# B&R Automation Studio project x20ost (part 2)

#### bnrcomserver.c
```c
/********************************************************************
 * COPYRIGHT -- Kontora
 ********************************************************************
 * Program: bnrmain
 * File: bnrlsens.c
 * Author: Abramenya
 * Created: January 19, 2009
 *******************************************************************/

#include "bnrcomserver.h"
#ifdef _DEFAULT_INCLUDES
 #include <AsDefault.h>
#endif
//extern SINT *chPortType[];
//extern SINT *chPortRate[];
extern WORD m_wPhoneKey;
extern char StrPhone[50];
/*
DEV_ARM_PORT_TCP=0,
DEV_ARM_PORT_UDP,
DEV_ARM_PORT_COM232,
DEV_ARM_PORT_COM458,
DEV_ARM_PORT_USB,
DEV_SYS_INTERFACE,
*/
SINT *chPortType[] =
{
	"TCP",
	"UDP",
	"RS232",
	"RS485",
	"USB",
};
SINT *chPortRate[] =
{
    "9600",
    "14400",
    "38400",
    "57600",
    "115200",
};
SINT *chPortParity[] =
{
    "N",
	"E",
	"O",
};
SINT *chPortData[] =
{
    "7",
	"8",
};
SINT *chPortStop[] =
{
    "1",
    "1.5",
    "2",
};
SINT *chTest = {"000=1.23000=2.30400=5.60005=192.10000=12334.20001=423.20001=4342.20"};
///char test={'000=0.00000=0.00000=0.00000=0.00000=0.00000=0.}
_GLOBAL UINT node_nr;
_GLOBAL UDINT status;
_GLOBAL CANopen_typ CANopen_01;
_GLOBAL CANnode_typ CANnode_01;
_GLOBAL  FRM_xopen_typ m_sXOpen;
_GLOBAL      XOPENCONFIG m_sConfig;
_GLOBAL      FRM_gbuf_typ m_sFrameBuff;
_GLOBAL      FRM_rbuf_typ m_sRBuff;
_GLOBAL      FRM_write_typ m_sSend;
_GLOBAL 	 FRM_read_typ m_sRecc;
_GLOBAL 	 FRM_close_typ m_sClose;
_GLOBAL 	 FRM_robuf_typ m_sRobuff;
#ifndef WIN32
_GLOBAL      FRM_mode_typ FrameModeStruct;
#endif
//USINT m_SendBuffer[300];
	 //USINT m_ReadBuffer[300];
#ifdef WIN32
#define  START_BYTE   0x7E
#define  STOP_BYTE    0xE7
#define  INVERSE_BYTE 0x55
CComServer *m_nCommServer;
BYTE m_byReadBuffer[300];
BYTE m_bySendBuffer[300];
HANDLE hCom;
OVERLAPPED  osReceive, osSend, osOverlap,osOverlapR;
COMSTAT  csStat;
HANDLE  hSendThread,hSendMsgThread,hReceiveThread,hMakeThread;
HANDLE  WaitEvents[2],evMake;
DWORD   dSendThreadId,dMakeThreadId,dSendMsgThreadId,dReceiveThreadId;
DWORD   dwThrdParam;
void RxCharProc(void);
static DWORD WINAPI SendRsThread(LPVOID lpCComm);
static DWORD WINAPI SendMsgThread(LPVOID lpCComm);
static DWORD WINAPI MakeThread(LPVOID lpCComm);
BOOL OpenPort(char *szComPort, DWORD dwBaud);
BOOL StartPort(char *szPortStr,DWORD dwBaud);
BOOL OpenPort(char *szComPort, DWORD dwBaud)
{
	DCB     dcb;
	COMMTIMEOUTS  ctCom;
	LPSTR lpMsgBuf;
	char  S[100];
	memset(&dcb,0,sizeof(DCB));
	dcb.DCBlength = sizeof(DCB);
    hCom = CreateFile(szComPort,
		GENERIC_READ | GENERIC_WRITE,
		0,
		NULL,
		OPEN_EXISTING,
		FILE_FLAG_OVERLAPPED,
		NULL);
    if (hCom == INVALID_HANDLE_VALUE)
		// ошибка открытия порта
    {
        FormatMessage(
            FORMAT_MESSAGE_ALLOCATE_BUFFER | FORMAT_MESSAGE_FROM_SYSTEM,
            NULL,
            GetLastError(),
            MAKELANGID(LANG_NEUTRAL, SUBLANG_DEFAULT), // Default language
            (LPTSTR) &lpMsgBuf,
            0,
            NULL
			);
        strcpy(S, "Error Opening. ");
        strcat(S, lpMsgBuf);
		printf("\n(__)Com::>%s",S);
		//Info("\n(__)Com::>%s",);
        //MessageBox(NULL, S, "RS232.Open", MB_OK);
        LocalFree( lpMsgBuf );
        return FALSE;
    }
    if (!GetCommState(hCom, &dcb))
		// ошибка получения параметров DCB
    {
        //MessageBox(NULL," Ошибка получения параметров DCB", "RS232.Open", MB_OK);
		printf("\n(__)Com::>Error Get Patrameters DCB");
        CloseHandle(hCom);
        return FALSE;
    }
    dcb.BaudRate = dwBaud;
    dcb.ByteSize = 8;
    dcb.Parity   = NOPARITY;
	//dcb.Parity   = EVENPARITY;
    dcb.StopBits = ONESTOPBIT;
	dcb.fDtrControl = DTR_CONTROL_HANDSHAKE;
	dcb.fRtsControl = RTS_CONTROL_HANDSHAKE;
    //dcb.EvtChar  = (CHAR)STOP_BYTE;
    if (!SetCommState(hCom, &dcb))
		// ошибка установки параметров DCB
    {
        //MessageBox(NULL," Ошибка установки параметров DCB", "RS232.Open", MB_OK);
		printf("\n(__)Com::>Error Create State DCB");
        CloseHandle(hCom);
        return FALSE;
    }
    ctCom.ReadIntervalTimeout = 10;
    ctCom.ReadTotalTimeoutMultiplier  = ctCom.ReadTotalTimeoutConstant  = 1;
    ctCom.WriteTotalTimeoutMultiplier = ctCom.WriteTotalTimeoutConstant = 1;
    if (!SetCommTimeouts(hCom, &ctCom))
		// ошибка установки параметров COMMTIMEOUTS
    {
        //MessageBox(NULL," Ошибка установки параметров COMMTIMEOUTS", "RS232.Open", MB_OK);
		printf("\n(__)Com::>Error DCB");
        CloseHandle(hCom);
        return FALSE;
    }
    //if (!SetCommMask(hCom, EV_RXCHAR|EV_TXEMPTY))
	if (!SetCommMask(hCom, EV_TXEMPTY))
		//    if (!SetCommMask(hCom, EV_BREAK | EV_RXCHAR))
		// ошибка установки маски событий
    {
		printf("\n(__)Com::>Error Create Mask Events");
        CloseHandle(hCom);
        return FALSE;
    }
    PurgeComm(hCom, PURGE_TXCLEAR | PURGE_RXCLEAR);
    // COM-порт успешно открыт и инициализирован
    return TRUE;
}
BOOL StartPort(char *szPortStr,DWORD dwBaud)
{
	if (OpenPort(szPortStr, dwBaud) != TRUE)
	{
		return FALSE;
	}
	if ((osOverlap.hEvent = CreateEvent(NULL, FALSE, FALSE, NULL)) == NULL)
	{
		printf("\n(__)Com::> Error Create osOverlap.hEvent");
		return FALSE;
	}

	if ((osReceive.hEvent = CreateEvent(NULL, FALSE, FALSE, NULL)) == NULL)
	{
		printf("\n(__)Com::> Error Create osReceive.hEvent");
		return FALSE;
	}
	if ((osSend.hEvent = CreateEvent(NULL, FALSE, FALSE, NULL)) == NULL)
	{
		printf("\n(__)Com::> Error Create osSend.hEvent");
		return FALSE;
	}
	if ((evMake = CreateEvent(NULL, FALSE, FALSE, NULL)) == NULL)
	{
		printf("\n(__)Com::> Error Create evMake");
		return FALSE;
	}
	if ((hMakeThread = CreateThread(NULL,0,MakeThread,&dwThrdParam,0,&dMakeThreadId)) == NULL)
	{
		printf("\n(__)Com::> Error Create hMakeThread");
		return FALSE;
	}
	if ((hSendThread = CreateThread(NULL,0,SendRsThread,&dwThrdParam,0,&dSendThreadId)) == NULL)
	{
		printf("\n(__)Com::> Error Create hReceiveThread");
		return FALSE;
	}

	if ((hSendMsgThread = CreateThread(NULL,0,SendMsgThread,&dwThrdParam,0,&dSendMsgThreadId)) == NULL)
	{
		printf("\n(__)Com::> Error Create hSensMsgThread");
		return FALSE;
	}
	SetThreadPriority(hSendThread, THREAD_PRIORITY_HIGHEST);
	SetThreadPriority(hSendMsgThread, THREAD_PRIORITY_NORMAL);
	SetThreadPriority(hMakeThread, THREAD_PRIORITY_NORMAL);
	ResumeThread(hSendThread);
	ResumeThread(hSendMsgThread);
	ResumeThread(hMakeThread);
	return TRUE;
}
void ClosePort(void)
{
    if (hCom != INVALID_HANDLE_VALUE)
    {
      CloseHandle(hCom);
      hCom = INVALID_HANDLE_VALUE;
    }
}
DWORD WINAPI SendMsgThread(LPVOID lpCComm)
{
    while(1)
    {
      m_nCommServer->SendThread(m_nCommServer);
	  Sleep(100);
    }
}
DWORD WINAPI SendRsThread(LPVOID lpCComm)
{
	DWORD dwMask,dwBytesTrans;
	//SMESSAGE mMsg;
	while(1)
	{
      //printf("\n(__)Com::>SendRsThread");
	  WaitCommEvent(hCom,&dwMask,&osOverlap);
	  //switch (WaitForSingleObject(osOverlap.hEvent,INFINITE))
	  switch (WaitForSingleObject(osOverlap.hEvent,5000))
	  {
	    case WAIT_OBJECT_0:
			 if (GetOverlappedResult(hCom,&osOverlap,&dwBytesTrans,TRUE))
			 {
               if (dwMask&EV_TXEMPTY)
               {
                //printf("\n(__)Com::>EV_TXEMPTY");
				m_sSend.status = 0;
				m_nCommServer->m_StatusWrite = 0;
               }
			   if (dwMask&EV_RXCHAR)
               {
				//printf("\n(__)Com::>EV_RXCHAR");
				//m_nCommServer->ReceiveThread(m_nCommServer);
				//RxCharProc();
               }
			 }
	  	break;
		case WAIT_TIMEOUT:
			 m_sSend.status = 0;
			 m_nCommServer->m_StatusWrite = 0;
			 PurgeComm(hCom, PURGE_TXCLEAR | PURGE_RXCLEAR);
			 //printf("\n(__)Com::>TX:WAIT_TIMEOUT");
		break;
	  }
	  //Sleep(1);
	}
}
void FRM_xopen(FRM_xopen_typ *pType)
{
    StartPort("COM4",1200);
};
void FRM_close(FRM_close_typ *pType){};
void FRM_gbuf(FRM_gbuf_typ *pType)
{
	pType->status = 0;
	pType->buflng = 300;
	pType->buffer = &m_bySendBuffer[0];
};
void FRM_rbuf(FRM_rbuf_typ *pType){};
void FRM_robuf(FRM_robuf_typ *pType){};
char chBuff[100];
void FRM_write(FRM_write_typ *pType)
{
	DWORD dwSentBytes;
	BOOL res;
	pType->status = 1;
	m_nCommServer->m_StatusWrite = 1;
	if(!WriteFile(hCom, pType->buffer, pType->buflng, &dwSentBytes,&osSend))
	//strcpy(chBuff,"Abramenya Alex");
	//if(!WriteFile(hCom, chBuff, strlen(chBuff), &dwSentBytes,&osOverlap))
    {
     if(GetLastError() != ERROR_IO_PENDING)
     {
	  // Ошибка записи данных
      res = FALSE;
	  printf("\n(__)Com::>Write Error 0.");
     }else
     {
      if(!GetOverlappedResult(hCom, &osSend, &dwSentBytes, TRUE))
      {
	   printf("\n(__)Com::>Write Error 1.");
      }else
      {
	   // Запись данных закончена
       res = TRUE;
	   //pType->status = 1;
	   //m_nCommServer->m_StatusWrite = 1;
	   //printf("\n(__)Com::>Write Ok 0.");
      }
     }
    }
    else
    {
	 // Запись успешно завершена
     res = TRUE;
	 //printf("\n(__)Com::>Write Ok 1.");
    }
};
BYTE pb_mBoxDoRead[5000];
BYTE pb_mBoxRead[3000];
BYTE pb_mBoxCont[5000];
WORD w_mBoxSize  = 0x7ff;
WORD w_mBoxCSize = 0x7ff;
WORD w_mBoxWrite = 0;
WORD w_mBoxRead  = 0;
WORD w_mBoxMesCt = 0;
//WORD w_mBoxSEnd  = 50000;
WORD mCurLen=0;
WORD m_sSize=0;
WORD w_lLength=0;
void MakeMessage(void);
void CopyMessage(WORD wLen);
/*
Success := ReadFile(FHandle, pb_mBoxDoRead, w_lLength, BytesTrans, @Ov);
		 for i:=0 to w_lLength-1 do
		 Begin
		  pb_mBoxCont[w_mBoxWrite]:=pb_mBoxDoRead[i];
          w_mBoxWrite := (w_mBoxWrite + 1) and BSZ;
		  //SendDebug('(__)Synchro Buffer NULL.');
		 End;

			 //SendDebug('(__)RD::');
			 //for i:=0 to w_lLength-1 do SendDebug(' '+IntToStr(pb_mBoxCont[i]));
			 //Success := Success and GetOverlappedResult(FHandle, Ov, BytesTrans, False);
			 //w_mBoxWrite := (w_mBoxWrite + w_lLength)and $7ff;
w_mBoxSize  := w_mBoxSize   - w_lLength;
m_sSize     := w_mBoxCSize  - w_mBoxSize;
			 if ((pb_mBoxCont[w_mBoxRead]=$68)or(pb_mBoxCont[w_mBoxRead]=$10)) then
				 Begin
m_byMType := 0;
			 SetEvent(hRxEvent);
			 End else
				 Begin
m_byMType  := 1;
w_mBoxSize  := BSZ;
w_mBoxCSize := BSZ;
w_mBoxWrite := 0;
w_mBoxRead  := 0;
w_mBoxMesCt := 0;
m_sSize:=0;
FBlTxEmpty := True;
			SendDebug('(__)Synchro Buffer.');
			//SetEvent(hRxEvent);
  End;
*/
void FRM_read(FRM_read_typ *pType)
{
	DWORD Errors,BytesTrans;
	BYTE i;
	ClearCommError(hCom, &Errors, &csStat);
	pType->status = 1;
	if (csStat.cbInQue!=0)
	{
	 pType->buffer = &m_byReadBuffer[0];
	 w_lLength = csStat.cbInQue;
     if(ReadFile(hCom, pType->buffer, w_lLength, &BytesTrans, &osReceive))
	 //if(ReadFile(hCom, m_byReadBuffer, w_lLength, &BytesTrans, &osReceive))
	 {
	  //for(i=0;i<w_lLength-1;i++)printf(" %x",m_byReadBuffer[i]);
	  pType->buflng = w_lLength;
	  pType->status = 0;
	 }else Info("\nError Read_0.");
	}
}
void RxCharProc(void)
{
	DWORD Errors,BytesTrans,dwB;
    BOOL  res;
	INT   i,wI,lLen;
	ClearCommError(hCom, &Errors, &csStat);
	if (csStat.cbInQue!=0)
	{
     w_lLength = csStat.cbInQue;
     if ((w_lLength<=0)||(w_lLength>500)) return;
     wI = w_mBoxWrite;
     if((wI+w_lLength)<=w_mBoxCSize)res = ReadFile(hCom, &pb_mBoxCont[wI], w_lLength, &BytesTrans, &osReceive);else
	 {
      res = ReadFile(hCom, &pb_mBoxDoRead[0], w_lLength, &BytesTrans, &osReceive);
	  for (i=0;i<w_lLength;i++){pb_mBoxCont[wI]=pb_mBoxDoRead[i];wI = (wI + 1) & 0x7ff;}
	 }
	 if(GetOverlappedResult(hCom, &osReceive, &dwB, TRUE))
	 {
	  //printf("\n(__)COM::>");for(i=0;i<w_lLength;i++)printf(" %x",pb_mBoxCont[w_mBoxWrite+i]);

	  w_mBoxWrite = (w_mBoxWrite + w_lLength)& 0x7ff;
      mCurLen=mCurLen+w_lLength;
      w_mBoxSize  = w_mBoxSize  - w_lLength;
	  if ((pb_mBoxCont[w_mBoxRead]==0x68)||(pb_mBoxCont[w_mBoxRead]==0x10))
	  {
       m_sSize=w_mBoxCSize-w_mBoxSize;
       SetEvent(evMake);
	   mCurLen=0;
	  }

	 }else printf("\n(__)Com::>RxRead Error.");
	}
}
void MakeMessage(void)
{
   WORD lLen,i;
   //printf("\n(__)COM::>MAKE_M:%x",pb_mBoxCont[w_mBoxRead]);
   lLen = pb_mBoxCont[(w_mBoxRead+1) & 0x7ff];
   while((m_sSize>=(lLen+6))&&(pb_mBoxCont[w_mBoxRead]==0x68))CopyMessage(lLen+6);
   lLen = 5;
   while((m_sSize>=lLen)&&(pb_mBoxCont[w_mBoxRead]==0x10))CopyMessage(lLen);
}
void CopyMessage(WORD wLen)
{
   INT i;
   SMESSAGE sMsg;
   for(i=0;i<wLen;i++)
   {
    pb_mBoxRead[i]=pb_mBoxCont[w_mBoxRead];
    w_mBoxSize++;
    w_mBoxRead=(w_mBoxRead+1)& 0x7ff;
   }
   m_sSize = (w_mBoxCSize-w_mBoxSize) & 0x7ff;
   m_sRecc.buflng = wLen;
   memcpy(&m_byReadBuffer[0],pb_mBoxRead, wLen);
   m_nCommServer->ReceiveThread(m_nCommServer);
   //printf("\n(__)COM::>");for(i=0;i<wLen;i++) printf(" %x",pb_mBoxRead[i]);
}
DWORD WINAPI MakeThread(LPVOID lpCComm)
{
	BYTE i;
	 while(1)
	 {
      WaitForSingleObject(evMake,INFINITE);
	  MakeMessage();
	  //printf("\n(__)COM::>MakeM.");
	 }
}
void CANopen(CANopen_typ *pCANOpen){};
void CANnode(CANnode_typ *pCANnode){};
#endif

void CComServer_Init(This,SARMINTERFACE *pArm)
{
    DECLARE_MULTI_OPEN(CComServer,CCyclicSystem)
    #ifdef WIN32
	m_nCommServer = pT;
    #endif
	pT->m_pArm = pArm;
	FDEFINE(DEV_RSMMD_BOX_ID,DEV_RSMMD_BOX_SZ);
	FDEFINE(DEV_RSBUF_BOX_ID,DEV_RSBUF_BOX_SZ);
	pB->SetBoxID(pB,DEV_RSMMD_BOX_ID);

	InitObject(CMTimer,&pT->m_nConnTMR);
	pT->m_nConnTMR.SetTimer(&pT->m_nConnTMR,DIR_PHTOPH,DIR_PHTOPH,EV_TMR_SRR_REQ,0,0,DEV_RSMMD_BOX_ID);
	//pT->m_nConnTMR.OnTimer(&pT->m_nConnTMR,10);
	pT->m_blMsgFind = FALSE;
	pT->m_byType = pArm->byType;
	pT->m_byRate = pArm->byPortRate;
	pT->InByteCount_DATA = 0;

	strcpy(pT->m_chStringMode, chPortType[pT->m_pArm->byType]);
	strcat(pT->m_chStringMode,", ");
	strcat(pT->m_chStringMode, chPortRate[pT->m_pArm->byPortRate]);
	strcat(pT->m_chStringMode,", ");
	strcat(pT->m_chStringMode, chPortParity[pT->m_pArm->stTcpAddr.byAddr0]);
	strcat(pT->m_chStringMode,", ");
	strcat(pT->m_chStringMode, chPortData[pT->m_pArm->stTcpAddr.byAddr1]);
	strcat(pT->m_chStringMode,", ");
	strcat(pT->m_chStringMode, chPortStop[pT->m_pArm->stTcpAddr.byAddr2]);

	strcpy(pT->m_chStringDevice, "SL0.IF1");
	#ifdef DEB_CComServer
	Info("\n(__)CTCPS::>Create %s.Device: %s Mode: %s",
	chPortType[pT->m_byType],pT->m_chStringDevice,pT->m_chStringMode);
	#endif
	pT->SynBuff(pT);
    pT->InitSRV(pT);
	//pT->m_nConnTMR.OnTimer(&pT->m_nConnTMR,200);
	pT->m_StatusWrite = 0;
	pT->m_bSrvState = DRV_ST_CONN;
	pT->m_bCliState = DRV_ST_CONN;
}
/*
if(pA->byA2==0) pR->byNumber          = (BYTE)pA->wParam; //Port Number
if(pA->byA2==1) pR->byType            = (BYTE)pA->wParam; //Port Type
if(pA->byA2==2) pR->byPortRate        = (BYTE)pA->wParam; //Port Rate
if(pA->byA2==3) pR->stTcpAddr.byAddr0 = (BYTE)pA->wParam; //Parity
if(pA->byA2==4) pR->stTcpAddr.byAddr1 = (BYTE)pA->wParam; //Data Bits
	 if(pA->byA2==5) pR->stTcpAddr.byAddr2 = (BYTE)pA->wParam; //Stop Bits
*/
void CComServer_SetPortSett(This)
{
    DECLARE_MULTI_OPEN(CComServer,CCyclicSystem)
    strcpy(pT->m_chStringDevice, "SL0.IF1");
	memset(pT->m_chStringNewMode,0,sizeof(pT->m_chStringNewMode));

	strcpy(pT->m_chStringNewMode, chPortType[pT->m_pArm->byType]);
	strcat(pT->m_chStringNewMode,", ");
	strcat(pT->m_chStringNewMode, chPortRate[pT->m_pArm->byPortRate]);
	strcat(pT->m_chStringNewMode,", ");
	strcat(pT->m_chStringNewMode, chPortParity[pT->m_pArm->stTcpAddr.byAddr0]);
	strcat(pT->m_chStringNewMode,", ");
	strcat(pT->m_chStringNewMode, chPortData[pT->m_pArm->stTcpAddr.byAddr1]);
	strcat(pT->m_chStringNewMode,", ");
	strcat(pT->m_chStringNewMode, chPortStop[pT->m_pArm->stTcpAddr.byAddr2]);
    #ifndef WIN32
    FrameModeStruct.ident  = m_sXOpen.ident;
    FrameModeStruct.mode   = (UDINT)pT->m_chStringNewMode;
    FrameModeStruct.enable = 1;
    FRM_mode(&FrameModeStruct);
    #endif
}
void CComServer_SynBuff(This)//CANOpen
{
    DECLARE_MULTI_OPEN(CComServer,CCyclicSystem)
	pT->w_mBoxSize  = BUFF_SZ;
    pT->w_mBoxCSize = BUFF_SZ;
	pT->w_mBoxWrite = 0;
	pT->w_mBoxRead  = 0;
	pT->m_sSize     = 0;
	pT->w_lLength   = 0;
	pT->w_lMsgLen   = 0;
	memset(&pT->pb_mBoxCont[0],0,10);
	#ifdef DEB_CComServer
	Info("\n(__)CTCPS::>Synchro.");
    #endif
}
_GLOBAL FRM_xopen_typ FrameXOpenStruct;
_GLOBAL XOPENCONFIG XOpenConfigStruct;
void CComServer_InitSRV(This)
{
    DECLARE_MULTI_OPEN(CComServer,CCyclicSystem)

	CANopen_01.enable    = 1;
    CANopen_01.baud_rate = 25;
    CANopen_01.cob_anz   = 5;
    CANopen_01.device    = 0;
    CANopen(&CANopen_01);

	//Server Init
    m_sConfig.idle     = 10;
    m_sConfig.delimc   = 0;
    m_sConfig.delim[0] = 0;
	m_sConfig.delim[1] = 0;
	m_sConfig.tx_cnt   = 2;
	m_sConfig.rx_cnt   = 2;
	m_sConfig.tx_len   = 256;
	m_sConfig.rx_len   = 256;
	m_sConfig.argc     = 0;
	m_sConfig.argv     = 0;

	strcpy(pT->m_chStringMode, "RS232, 57600, E, 8, 1");
	m_sXOpen.device    = (UDINT) pT->m_chStringDevice;
	m_sXOpen.mode      = (UDINT) pT->m_chStringMode;
    m_sXOpen.config    = (UDINT)&m_sConfig;
	m_sXOpen.enable    = 1;
	pT->m_StatusOpen   = 0;
    #ifndef WIN32
	pT->m_nConnTMR.OnTimer(&pT->m_nConnTMR,30);
    #else
	pT->m_nConnTMR.OnTimer(&pT->m_nConnTMR,30);
	//pT->Open(pT);
    #endif
}
_GLOBAL INT nOPEN,nCLOSE;

BOOL CComServer_Open(This)
{
    DECLARE_MULTI_OPEN(CComServer,CCyclicSystem)
	SHORTMESSAGE m_sMsg;

	CANnode_01.enable = 1;
    CANnode(&CANnode_01);
    node_nr = CANnode_01.node_nr;
    #ifdef WIN32
	node_nr = 1;
	//pT->m_StatusOpen = 0;
    #endif
    if((node_nr==1)&&(pT->m_StatusOpen==0))
	{
	FRM_xopen(&m_sXOpen);
	if(m_sXOpen.status==0)
	{
	 nOPEN++;
	 m_sRecc.ident      = m_sXOpen.ident;
	 m_sSend.ident      = m_sXOpen.ident;
	 m_sClose.ident     = m_sXOpen.ident;
	 m_sFrameBuff.ident = m_sXOpen.ident;
	 m_sRBuff.ident     = m_sXOpen.ident;
	 m_sRecc.buffer	    = (UDINT)&pT->m_ReadBuffer[0];
	 m_sSend.buffer     = (UDINT)&pT->m_SendBuffer[0];
	 m_sFrameBuff.buffer= m_sSend.buffer;
	 m_sRBuff.buffer    = m_sRecc.buffer;
	 m_sRecc.enable     = 1;
	 m_sSend.enable     = 1;
	 m_sClose.enable    = 1;
	 m_sFrameBuff.enable= 1;
	 m_sRBuff.enable    = 1;
	 pT->m_StatusOpen   = 1;
	 pT->m_StatusWrite  = 0;
     #ifdef IF_MODEM
	 SendCommand(PH_INIT_REQ,"AT+ipr=57600");
	 SendCommand(PH_INIT_REQ,"AT+icf=2,1");
	 SendCommand(PH_INIT_REQ,"AT+ifc=0,0");
	 SendCommand(PH_INIT_REQ,"AT&D1");
	 SendCommand(PH_INIT_REQ,"AT&C1");
	 //SendCommand(PH_INIT_REQ,"AT&S0");
	 SendCommand(PH_INIT_REQ,"ATS0=1");
	 SendCommand(PH_INIT_REQ,"AT+CLIP=1");
     #endif
	 pT->SendSMessage(pT,DEV_KPMDL_BOX_ID,DIR_PHTOKP,PH_CALL_REQ);
	 return TRUE;
	}
 	}
	if((node_nr==3)&&(pT->m_StatusOpen==1))
	{
	  nCLOSE++;
	  pT->m_StatusOpen = 0;
      pT->Close(pT);
	  return TRUE;
	}
	return FALSE;
}
void CComServer_Enable(This)
{
	DECLARE_MULTI_OPEN(CComServer,CCyclicSystem)
	m_sXOpen.enable = 1;
}
void CComServer_Disable(This)
{
	DECLARE_MULTI_OPEN(CComServer,CCyclicSystem)
	m_sXOpen.enable = 0;
}
void CComServer_Close(This)
{
    DECLARE_MULTI_OPEN(CComServer,CCyclicSystem)
	m_sClose.enable = 1;
	FRM_close(&m_sClose);
}
BOOL CComServer_SendMessage(This,SMESSAGE *pMsg)
{
	DECLARE_MULTI_OPEN(CComServer,CCyclicSystem)
	BOOL res = TRUE;
	if(pT->m_StatusOpen==1)
	{
	 FRM_gbuf(&m_sFrameBuff);
     m_sSend.buflng = pMsg->m_swLen-9;
	 memcpy(m_sSend.buffer, &pMsg->m_sbyInfo[0],m_sSend.buflng);
	 FRM_write(&m_sSend);
	 pT->m_StatusWrite  = m_sSend.status;
	 if(pT->m_StatusWrite==0) res = TRUE;else res = FALSE;
	}
	return res;
}
_GLOBAL INT nSND;
_GLOBAL INT nSendThread;
void CComServer_SendThread(This)
{
    DECLARE_MULTI_OPEN(CComServer,CCyclicSystem)
	nSendThread++;
    //if(pT->m_StatusWrite==0)
	if(pT->m_StatusOpen==1)
    {
	 #ifdef DEB_CComServer
	 //pT->TestMsg(pT);
     #endif
	 if(FGET(DEV_RSBUF_BOX_ID,&pT->m_sMsg))
	 {
	  //Info("\n(__)CRSSM::>TX:%M",&pT->m_sMsg);
	  if(pT->m_sMsg.m_swLen<=256)
	  {
	   nSND++;
       pT->SendMessage(pT,&pT->m_sMsg);
	  }//else
	    //Info("\n(__)CRSSM::>Wery Long Message!");
	 }
	}
}
_GLOBAL INT nGETL1;
BOOL CComServer_GetMessage(This,SMESSAGE *pMsg)
{
    DECLARE_MULTI_OPEN(CComServer,CCyclicSystem)
	BYTE i,*pBuff;
	BOOL res=FALSE;
	SMESSAGE csM;
	if(pT->m_StatusOpen==1)
	{
	FRM_read(&m_sRecc);
	pT->m_StatusRead       = m_sRecc.status;
	if(pT->m_StatusRead==0)
	{
	 pT->m_ReadBufferLength = m_sRecc.buflng;
	 pBuff                  = m_sRecc.buffer;
	 /*
	 csM.m_sbyInfo[0] = 0x7e;
	 csM.m_sbyInfo[1] = 'A';
	 csM.m_sbyInfo[2] = 'l';
	 csM.m_sbyInfo[3] = 'e';
	 csM.m_sbyInfo[4] = 'x';
	 csM.m_sbyInfo[5] = 'a';
	 csM.m_sbyInfo[6] = 'n';
	 csM.m_sbyInfo[7] = 'd';
	 csM.m_sbyInfo[8] = 'e';
	 csM.m_sbyInfo[9] = 'r';
	 csM.m_sbyInfo[10] = 0xe7;
	 */

	 //memcpy(&csM.m_sbyInfo[0],m_sRecc.buffer,pT->m_ReadBufferLength);
	 //csM.m_swLen = 9 + pT->m_ReadBufferLength;
	 //Info("\n(__)CRSSM::>MSG:%M",&csM);

	 //m_sRBuff.buffer = m_sRecc.buffer;
	 //m_sRBuff.buflng = pT->m_ReadBufferLength;
	 //FRM_rbuf(&m_sRBuff);
	 //res = TRUE;
	 //nGETL1++;
	 //Info("\nMSG::>");
	 //csM.m_swLen = pT->m_ReadBufferLength+9;
	 for( i=0;i<pT->m_ReadBufferLength;i++)
	 {
	  pT->pb_mBoxCont[pT->w_mBoxWrite] = pBuff[i];
      //Info(" %b",&pT->pb_mBoxCont[pT->w_mBoxWrite]);
	  //printf(" %c",pT->pb_mBoxCont[pT->w_mBoxWrite]);
      pT->w_mBoxWrite = (pT->w_mBoxWrite + 1) & BUFF_SZ;
	 }
	 //FPUT(DEV_RSBUF_BOX_ID,(BYTE*)&csM);
	 pT->w_mBoxSize -= pT->m_ReadBufferLength;
	 pT->m_sSize     = pT->w_mBoxCSize-pT->w_mBoxSize;
	 //Info("\nRD::>%b PRD::>%w PWD::>%w FND::>%b",&pT->pb_mBoxCont[pT->w_mBoxRead],&pT->w_mBoxRead,&pT->w_mBoxWrite,&pT->m_blMsgFind);
	 //printf(" %c %c", pT->pb_mBoxCont[pT->w_mBoxRead],pT->pb_mBoxCont[pT->w_mBoxRead+1]);
	 //if ((pT->pb_mBoxCont[pT->w_mBoxRead]==0x3d)&&(pT->pb_mBoxCont[pT->w_mBoxRead+1]==0x30))
	 if ((pT->pb_mBoxCont[pT->w_mBoxRead]==0x3d))
	 {
	  pT->m_blMsgFind = TRUE;
	  if(res = pT->MakeMsgData(pT,pMsg))
	  {
	   pT->m_blMsgFind = FALSE;
	   res = TRUE;
	  }
	 }else
		 pT->SynBuff(pT);
	 //if (pT->m_blMsgFind==FALSE)
	 //{
	 //	pT->MakeTextMessage(pT);
 	 //}else /*if (pT->pb_mBoxCont[pT->w_mBoxRead]==0x41)*/ pT->SynBuff(pT);
	 m_sRBuff.buffer = m_sRecc.buffer;
	 m_sRBuff.buflng = pT->m_ReadBufferLength;
	 FRM_rbuf(&m_sRBuff);
     }
	}
	return res;
}
BOOL CComServer_MakeMsgData(This,SMESSAGE *pMsg)
{
    DECLARE_MULTI_OPEN(CComServer,CCyclicSystem)
	WORD lLen,i,nCM=0;
	BOOL res = FALSE;
	lLen = 1;
	pT->w_lMsgLen = pT->w_lMsgLen + pT->m_ReadBufferLength;
	if (pT->w_lMsgLen>BUFF_SZ) {pT->SynBuff(pT);return res;}
    for (i=1;i<pT->w_lMsgLen-1;i++)
	{
	 lLen++;
	 if (pT->pb_mBoxCont[(pT->w_mBoxRead+i)& BUFF_SZ]==0x2e) nCM++;
	 if (nCM>1){pT->SynBuff(pT);return res;}
	 if (lLen>300) {pT->SynBuff(pT);return res;}
     if (pT->pb_mBoxCont[(pT->w_mBoxRead+i)& BUFF_SZ]==0x3d)
     {
	  pT->CopyMessage(pT,lLen,pMsg);
	  //pT->SynBuff(pT);
	  pT->w_lMsgLen = 0;
	  return TRUE;
	 }
	}
	return res;
}
BOOL CComServer_CopyMessage(This,WORD wLen,SMESSAGE *pMsg)
{
    DECLARE_MULTI_OPEN(CComServer,CCyclicSystem)
    INT i,j=0;BYTE byCRC;
	BOOL blCRC;
	for(i=0;i<wLen;i++)
	{
	 if ((i!=0)&&(i!=wLen-1)){pMsg->m_sbyInfo[j]=pT->pb_mBoxCont[pT->w_mBoxRead];j++;}
	 pT->w_mBoxSize =(pT->w_mBoxSize+1)& BUFF_SZ; ;
	 pT->w_mBoxRead=(pT->w_mBoxRead+1)& BUFF_SZ;
	 //Info(" %b",&pMsg->m_sbyInfo[i]);
	 //printf(" %x",pMsg->m_sbyInfo[i]);
	}
	pMsg->m_sbyInfo[j++] = 0x00;
	pT->w_mBoxRead=(pT->w_mBoxRead-1)& BUFF_SZ;
	pT->m_sSize = (pT->w_mBoxCSize-pT->w_mBoxSize) & BUFF_SZ;
	pMsg->m_swLen         = j+9;
	pMsg->m_sbyFrom       = DIR_PHMDL;
	pMsg->m_sbyFor        = DIR_PHTOMS;
	pMsg->m_sbyIntType    = 0;
	pMsg->m_sbyServerID   = 0;
	pMsg->m_sbyType       = PH_VS0_REQ;
	pMsg->m_sbyDirection  = 0;
	pMsg->m_sbySensor     = 0;
	//byCRC = pMsg->m_sbyInfo[pMsg->m_swLen-9-2];
    //if (pMsg->m_sbyInfo[0]==MSG_SHRT_CODE)
	//if (byCRC==pT->CreateCRC(pT,&pMsg->m_sbyInfo[1],2)) blCRC = TRUE;
	return TRUE;
}
_GLOBAL INT nReceiveThread;
void CComServer_ReceiveThread(This)
{
    DECLARE_MULTI_OPEN(CComServer,CCyclicSystem)
	nReceiveThread++;
	if(pT->GetMessage(pT,&pT->m_sMsg)==TRUE)
	{
	 //Info("\n(__)CRSSM::>RX:%M",&pT->m_sMsg);
	 //if ((pT->nWsCount++)%10==0)
	 FPUT(DEV_MSMDL_BOX_ID,(BYTE*)&pT->m_sMsg);
	 //FPUT(DEV_RSBUF_BOX_ID,(BYTE*)&pT->m_sMsg);
	}
}
void CComServer_MakeTextMessage(This)
{
	DECLARE_MULTI_OPEN(CComServer,CCyclicSystem)
    BYTE byInByte;
    while (pT->w_mBoxWrite!=pT->w_mBoxRead)
	{
     byInByte = pT->pb_mBoxCont[pT->w_mBoxRead];
     pT->w_mBoxRead = (pT->w_mBoxRead+1) & BUFF_SZ;
     if (pT->w_mBoxSize>pT->w_mBoxCSize){pT->SynBuff(pT);return;};
     pT->w_mBoxSize++;
     if (byInByte==0x0d)
	 {
	   if (pT->InByteCount_DATA>1)
	   pT->ATHandler(pT,&pT->pb_mBoxDoTextRead[0],pT->InByteCount_DATA);
       pT->InByteCount_DATA = 0;
	 }else
	 {
       pT->pb_mBoxDoTextRead[pT->InByteCount_DATA] = byInByte;
       if (pT->InByteCount_DATA>100) {pT->InByteCount_DATA=0;pT->SynBuff(pT);}
       pT->InByteCount_DATA++;
	 }
	}
}
void CComServer_ATHandler(This,USINT *pComm,WORD wLen)
{
    DECLARE_MULTI_OPEN(CComServer,CCyclicSystem)
    WORD i,i0,i1,j=0;
	//printf("\nAT_MSG::>");for (i=0;i<wLen;i++)printf(" %c",pComm[i]);
	if (wLen<100)
	{
	pComm[wLen] = 0;
	if(pT->FindText(pT,"CONNECT",pComm)>0)
	{
     #ifdef DEB_CComServer
	 Info("\n(__)CRSSM::>CONNECT 9600");
     #endif
	 pT->Connect(pT);
	 return;
	}
	if(pT->FindText(pT,"NO CAR",pComm)>0)
	{
     #ifdef DEB_CComServer
	 Info("\n(__)CRSSM::>NO CARRIER");
     #endif
	 pT->Disconnect(pT);
	 return;
	}
	if(pT->FindText(pT,"+CLIP:",pComm)>0)
	{
     #ifdef DEB_CComServer
	 Info("\n(__)CRSSM::>+CLIP");
     #endif
     m_wPhoneKey = 0;
	 i0 = pT->FindText(pT," ",pComm);i1 = pT->FindText(pT,",",pComm);
     //printf("\nAT_PHO::>");
	 for (i=i0+2;i<i1-1;i++)
	 {
	  if (i>30) return;
	  m_wPhoneKey = m_wPhoneKey + ((pComm[i]&0x0f)+j);
	  //StrPhone[j]=pComm[i];
	  j++;
      //printf(" %c",pComm[i]);
	 }
	 return;
	}
	}else pT->SynBuff(pT);
}
INT CComServer_FindText(This,SINT *pSrc,SINT *pChar)
{
    DECLARE_MULTI_OPEN(CComServer,CCyclicSystem)
	WORD i,wSrcSumm=0,wLen,wStrLen;
	wLen    = strlen(pSrc);
	wStrLen = strlen(pChar);
	wSrcSumm = pT->CalckSumm(pT,(BYTE*)pSrc,wLen);
	for (i=0;i<wStrLen-wLen;i++)
	{
	 if (wSrcSumm==pT->CalckSumm(pT,(BYTE*)&pChar[i],wLen))
	 return i;
	}
	return -1;
}
WORD CComServer_CalckSumm(This,BYTE *pCH,WORD wLen)
{
    DECLARE_MULTI_OPEN(CComServer,CCyclicSystem)
	WORD i,wSrcSumm=0;
	for (i=0;i<wLen;i++)
	wSrcSumm += pCH[i];
    return wSrcSumm;
}
BYTE CComServer_CreateCRC(This,BYTE *pMsg,BYTE byLen)
{
	DECLARE_MULTI_OPEN(CComServer,CCyclicSystem)
	BYTE i,sum = 0;
	for(i=0;i<=byLen-1;i++)sum += pMsg[i];
	return sum;
}
_GLOBAL INT nRSEventHandler,nCheckOpen,nWatchOpen;
BOOL CComServer_EventHandler(This,SMESSAGE *pMsg)
{
    DECLARE_MULTI_OPEN(CComServer,CCyclicSystem)
	switch(pMsg->m_sbyFor)
	{
	  case DIR_101TOPH:
	       #ifdef DEB_CComServer
		   //Info("\n(__)CRSSM::>OUTP::%M",pMsg);
		   #endif
		   FPUT(DEV_RSBUF_BOX_ID,pMsg);
	  break;
	  case DIR_KPTO101:
	       nRSEventHandler++;
		   if(pMsg->m_sbyType==PH_CONN_REQ)
		   {
            #ifndef IF_MODEM
		    pT->Connect(pT);
            #else
		    FPUT(DEV_RSBUF_BOX_ID,pMsg);
            #endif
		   }
		   if((pMsg->m_sbyType==PH_DISC_REQ)||(pMsg->m_sbyType==PH_DISC0_REQ))
		   {
			//pT->Disconnect(pT);
			FPUT(DEV_RSBUF_BOX_ID,pMsg);
		   }
		   if(pMsg->m_sbyType==PH_INIT_REQ)
		   FPUT(DEV_RSBUF_BOX_ID,pMsg);
	  break;
	  case DIR_PHTOPH:
	       if (pMsg->m_sbyType==EV_TMR_SRR_REQ)
		   {
		   	//if(pT->m_StatusOpen==0)
			{
			 nCheckOpen++;
 		     pT->Open(pT);
			}
			pT->m_nConnTMR.OnTimer(&pT->m_nConnTMR,30);
		   }
	  break;
      case DIR_KPTOPH:
	       if (pMsg->m_sbyType==PH_CLOSE_PORT_REQ)
		   {
            //pT->Close(pT);
		   }
		   if(pMsg->m_sbyType==PH_INIT_PORT_REQ)
		   {
             pT->SetPortSett(pT);
		   }
	  break;
	  default:
	  break;
	}
	return TRUE;
}
void CComServer_Connect(This)
{
    DECLARE_MULTI_OPEN(CComServer,CCyclicSystem)
    SHORTMESSAGE m_sMsg;
	m_sMsg.m_swLen        = 9;
	m_sMsg.m_sbyFrom      = DIR_PHMDL;
	m_sMsg.m_sbyFor       = DIR_PHTO101P;
	m_sMsg.m_sbyIntType   = 0;
	m_sMsg.m_sbyServerID  = 0;
	m_sMsg.m_sbyType      = PH_CONN_IND;
	m_sMsg.m_sbyDirection = 0;
	m_sMsg.m_sbySensor    = 0;
	FPUT(DEV_101MD_BOX_ID,(BYTE*)&m_sMsg);
    #ifdef DEB_CComServer
	Info("\n(__)CRSSM::>OUTT::%M",&m_sMsg);
    #endif
}
void CComServer_SendSMessage(This,BYTE byBox,BYTE byFor,BYTE byType)
{
    DECLARE_MULTI_OPEN(CComServer,CCyclicSystem)
    SHORTMESSAGE m_sMsg;
	m_sMsg.m_swLen        = 9;
	m_sMsg.m_sbyFrom      = DIR_PHMDL;
	m_sMsg.m_sbyFor       = byFor;
	m_sMsg.m_sbyIntType   = 0;
	m_sMsg.m_sbyServerID  = 0;
	m_sMsg.m_sbyType      = byType;
	m_sMsg.m_sbyDirection = 0;
	m_sMsg.m_sbySensor    = 0;
	FPUT(byBox,(BYTE*)&m_sMsg);
    #ifdef DEB_CComServer
	Info("\n(__)CRSSM::>OUTT::%M",&m_sMsg);
    #endif
}
void CComServer_Disconnect(This)
{
    DECLARE_MULTI_OPEN(CComServer,CCyclicSystem)
    SHORTMESSAGE m_sMsg;
	m_sMsg.m_swLen        = 9;
	m_sMsg.m_sbyFrom      = DIR_PHMDL;
	m_sMsg.m_sbyFor       = DIR_PHTO101P;
	m_sMsg.m_sbyIntType   = 0;
	m_sMsg.m_sbyServerID  = 0;
	m_sMsg.m_sbyType      = PH_DISC_IND;
	m_sMsg.m_sbyDirection = 0;
	m_sMsg.m_sbySensor    = 0;
	FPUT(DEV_101MD_BOX_ID,(BYTE*)&m_sMsg);
    #ifdef DEB_CComServer
	Info("\n(__)CRSSM::>OUTT::%M",&m_sMsg);
    #endif
}
/*
12	12:58:38	hypertrm.exe	IRP_MJ_READ	Serial2	TIMEOUT	Length 14: 30 30 3D 30 2E 30 30 30 30 30 3D 30 2E 30
13	12:58:38	hypertrm.exe	IRP_MJ_READ	Serial2	TIMEOUT	Length 14: 30 30 30 30 3D 30 2E 30 30 30 30 30 3D 30
14	12:58:39	hypertrm.exe	IRP_MJ_READ	Serial2	TIMEOUT	Length 14: 2E 30 30 30 30 30 3D 30 2E 30 30 30 30 30
15	12:58:39	hypertrm.exe	IRP_MJ_READ	Serial2	TIMEOUT	Length 14: 3D 30 2E 30 30 30 30 30 3D 30 2E 30 30 30
16	12:58:39	hypertrm.exe	IRP_MJ_READ	Serial2	TIMEOUT	Length 14: 30 30 3D 30 2E 30 30 30 30 30 3D 30 2E 30
17	12:58:39	hypertrm.exe	IRP_MJ_READ	Serial2	TIMEOUT	Length 14: 30 30 30 30 3D 30 2E 30 30 30 30 30 3D 30
18	12:58:39	hypertrm.exe	IRP_MJ_READ	Serial2	TIMEOUT	Length 14: 2E 30 30 30 30 30 3D 30 2E 30 30 30 30 30
19	12:58:39	hypertrm.exe	IRP_MJ_READ	Serial2	TIMEOUT	Length 14: 3D 30 2E 30 30 30 30 30 3D 30 2E 30 30 30
20	12:58:40	hypertrm.exe	IRP_MJ_READ	Serial2	TIMEOUT	Length 14: 30 30 3D 30 2E 30 30 30 30 30 3D 30 2E 30
21	12:58:40	hypertrm.exe	IRP_MJ_READ	Serial2	TIMEOUT	Length 14: 30 30 30 30 3D 30 2E 30 30 30 30 30 3D 30
*/
void CComServer_TestMsg(This)
{
    DECLARE_MULTI_OPEN(CComServer,CCyclicSystem)
	SMESSAGE m_sMsg;
	m_sMsg.m_swLen        = 9+strlen(chTest);
	m_sMsg.m_sbyFrom      = DIR_PHMDL;
	m_sMsg.m_sbyFor       = DIR_101TOPH;
	m_sMsg.m_sbyIntType   = 0;
	m_sMsg.m_sbyServerID  = 0;
	m_sMsg.m_sbyType      = PH_DATA_RES;
	m_sMsg.m_sbyDirection = 0;
	m_sMsg.m_sbySensor    = 0;
	strcpy(&m_sMsg.m_sbyInfo[0],chTest);
	FPUT(DEV_RSMMD_BOX_ID,(BYTE*)&m_sMsg);
    #ifdef DEB_CComServer
	//Info("\n(__)CRSSM::>TEST::%M",&m_sMsg);
    #endif
}
void CComServer_CyclicProc(This)
{
    DECLARE_MULTI_OPEN(CComServer,CCyclicSystem)
	pT->ReceiveThread(pT);
	#ifndef WIN32
	pT->SendThread(pT);
	#endif
}
void CComServer_CComServer(This)
{
    DECLARE_MULTI_OPEN(CComServer,CCyclicSystem)
	DECLARE_REGISTRATION(CComServer,Init)
	DECLARE_REGISTRATION(CComServer,InitSRV)
	DECLARE_REGISTRATION(CComServer,SendMessage)
	DECLARE_REGISTRATION(CComServer,GetMessage)
    DECLARE_REGISTRATION(CComServer,Close)
	DECLARE_REGISTRATION(CComServer,Disable)
	DECLARE_REGISTRATION(CComServer,Enable)
	DECLARE_REGISTRATION(CComServer,Open)
	DECLARE_REGISTRATION(CComServer,ReceiveThread)
	DECLARE_REGISTRATION(CComServer,SendThread)
	DECLARE_REGISTRATION(CComServer,SynBuff)
	DECLARE_REGISTRATION(CComServer,MakeMsgData)
	DECLARE_REGISTRATION(CComServer,MakeTextMessage)
	DECLARE_REGISTRATION(CComServer,ATHandler)
	DECLARE_REGISTRATION(CComServer,CopyMessage)
	DECLARE_REGISTRATION(CComServer,CreateCRC)
	DECLARE_REGISTRATION(CComServer,Connect)
	DECLARE_REGISTRATION(CComServer,Disconnect)
	DECLARE_REGISTRATION(CComServer,FindText)
	DECLARE_REGISTRATION(CComServer,CalckSumm)
	DECLARE_REGISTRATION(CComServer,SendSMessage)
	DECLARE_REGISTRATION(CComServer,SetPortSett)
	DECLARE_REGISTRATION(CComServer,TestMsg)
	DECLARE_VIRTUAL_FUNC(CComServer,EventHandler)
	DECLARE_VIRTUAL_FUNC(CComServer,CyclicProc)
}

void CComServer_DCComServer(This)
{
	DECLARE_MULTI_OPEN(CComServer,CCyclicSystem)
	//DESTROY
}

DECLARE_MULTI_CREATE(CComServer,CCyclicSystem)
```

#### bnrconfig.c
```c
/********************************************************************
 * COPYRIGHT -- Kontora
 ********************************************************************
 * Program: bnrmain
 * File: bnrconfig.h
 * Author: Abramenya
 * Created: February 04, 2009
 *******************************************************************/
#ifndef WIN32
#include <bur/plctypes.h>
#endif
#include "typedefs.h"
#include "bnrmessage.h"
/*
REAL m_rlDy;
REAL m_rlKp;
REAL m_rlTn;
REAL m_rlKw;
REAL m_rlKfbk;
INT16 m_rlA;
	INT16 m_rlYman;
*/
#define PID_PARAM 20.0,0.4,6000.0,1.0,1.0,0,0
IMPORT_STATELIST(STL_LV00_SENS);//2-Out
IMPORT_STATELIST(STL_PS00_SENS);//2-Out
IMPORT_STATELIST(STL_TM00_SENS);//1-Out
IMPORT_STATELIST(STL_LV04_SENS);//1-Out
IMPORT_STATELIST(STL_LVN4_SENS);//0-Out
IMPORT_STATELIST(STL_PS04_SENS);//1-Out
//Digital Sensor Section
IMPORT_STATELIST(STL_DIGS00_SENS);//12-In 32-Out
SOUTGATE     nOutGateDF = {0,5100,11,60,0.0,1.0,NO,SDIR,NO,SMART_GTE,SL00,PN00,"п.xxx"};//Lev
#if MYSYSTEM_ID == 0
SINPUTGATE nINGT = {10,{
{496,100, 0,  95,  20,  70,  30, 70, 1.0,2.0,20000.0 ,1.0,1.0,1000.0 ,550.0 ,0,0,0,0,BASE_GTE,MAX_GTE,0,SL02,PN00,SNS_SMART,P_LEVEL,ST_OPEN,ST_OPEN,SNS_MD_AUTO},
{484,100, 0,  95,  20,  70,  30, 70, 1.0,2.0,20000.0 ,1.0,1.0,1000.0 ,550.0 ,0,0,0,0,BASE_GTE,MAX_GTE,1,SL02,PN01,SNS_SMART,P_LEVEL,ST_OPEN,ST_OPEN,SNS_MD_AUTO},
{480, 60, 0,  28,  20,  22,  21, 22, 0.0,3.0,250000.0,1.0,1.0,20400.0,600.0 ,0,0,0,0,BASE_GTE,MAX_GTE,2,SL02,PN02,SNS_SMART,P_PRESS,ST_OPEN,ST_OPEN,SNS_MD_AUTO},
{485,200, 0, 155, 145, 150, 145,150, 0.0,1.9,90000.0 ,1.0,1.0,1000.0 ,500.0 ,0,0,0,0,BASE_GTE,MAX_GTE,3,SL02,PN03,SNS_SMART,P_TEMPR,ST_OPEN,ST_OPEN,SNS_MD_AUTO},
{485,200, 0, 155, 145, 150, 145,150, 1.0,1.0,45000.0 ,1.0,1.0,1000.0 ,550.0 ,0,0,0,0,BASE_GTE,MAX_GTE,4,SL02,PN04,SNS_SMART,P_TEMPR,ST_OPEN,ST_OPEN,SNS_MD_AUTO},
{496,200, 0, 195, 185, 190, 185,190, 1.0,1.0,45000.0 ,1.0,1.0,1000.0 ,550.0 ,0,0,0,0,BASE_GTE,MAX_GTE,5,SL02,PN05,SNS_IDLES,P_TEMPR,ST_OPEN,ST_OPEN,SNS_MD_AUTO},
{496,200, 0, 195, 185, 190, 185,190, 0.0,1.0,90000.0 ,1.0,1.0,1000.0 ,500.0 ,0,0,0,0,BASE_GTE,MAX_GTE,6,SL02,PN06,SNS_SMART,P_TEMPR,ST_OPEN,ST_OPEN,SNS_MD_AUTO},
{496,200, 0, 195, 185, 190, 185,190, 1.0,1.0,45000.0 ,1.0,1.0,1000.0 ,550.0 ,0,0,0,0,BASE_GTE,MAX_GTE,7,SL02,PN07,SNS_SMART,P_TEMPR,ST_OPEN,ST_OPEN,SNS_MD_AUTO},
{485,200, 0, 155, 145, 150, 145,150, 1.0,1.0,45000.0 ,1.0,1.0,1000.0 ,550.0 ,0,0,0,0,BASE_GTE,MAX_GTE,8,SL03,PN00,SNS_SMART,P_TEMPR,ST_OPEN,ST_OPEN,SNS_MD_AUTO},
{496,200, 0, 195, 185, 190, 185,190, 1.0,1.0,45000.0 ,1.0,1.0,1000.0 ,550.0 ,0,0,0,0,BASE_GTE,MAX_GTE,9,SL03,PN01,SNS_SMART,P_TEMPR,ST_OPEN,ST_OPEN,SNS_MD_AUTO},
}};
SOUTPUTGATE nOTGT = {10,{
{0,5100,10,30,0.0,0.4,NZ,SDIR,0,SMART_GTE,SL04,PN02,"п.812/1"},//Lev LE1 RP4
{0,5100,15,30,0.0,0.4,NZ,SINV,0,SMART_GTE,SL04,PN03,"п.812/2"},//Lev LE1 RP3
{0,5100,20,30,0.2,1.0,NO,SDIR,0,SMART_GTE,SL04,PN00,"п.811/1"},//Prs PE1 RP2
{0,5100,25,30,0.2,0.8,NZ,SINV,0,SMART_GTE,SL04,PN01,"п.811/2"},//Prs PE1 RP1
{0,5100,30,30,0.2,1.0,NZ,SDIR,0,IDLES_GTE,SL04,PN05,"п.814"},  //Tmp TE1 RP5
{0,5100,35,30,0.2,1.0,NZ,SINV,0,IDLES_GTE,SL04,PN04,"п.815"},  //Tmp TE2 RP6
{0,5100,40,30,0.2,1.0,NZ,SDIR,0,IDLES_GTE,SL04,PN06,"п.813"},  //Tmp TE4 RP8
{0,5100,45,30,0.0,1.0,NO,SDIR,0,IDLES_GTE,SL05,PN00,"п.854"},  //Tmp TE5 RP10
{0,5100,50,30,0.0,1.0,NO,SDIR,0,IDLES_GTE,SL05,PN01,"п.855"},  //Tmp TE6 RP9
{0,5100,55,30,0.2,1.0,NZ,SDIR,0,IDLES_GTE,SL04,PN07,"п.511"},  //Tmp TE7 RP7
}};
SSOFTSWITCHTABLE  nSoftSwitchTable=
{
 0,"Switching Table For System AC-1",1,
 {
	//Switching For Direction 0
	{
      0,0,11,&nINGT,&nOTGT,
	  {
		{0 ,&nINGT.mIn[1], STL_LV00_SENS, SWC_CMD_SMR_CON,  TRUE, 1,{&nOTGT.mOut[0]}}, //LE
		{1 ,&nINGT.mIn[1], STL_LV00_SENS, SWC_CMD_SMR_CON,  TRUE, 1,{&nOTGT.mOut[1]}}, //LE
		{2 ,&nINGT.mIn[2], STL_PS00_SENS, SWC_CMD_SMR_CON,  TRUE, 1,{&nOTGT.mOut[2]}}, //PE1 Out0
		{3 ,&nINGT.mIn[2], STL_PS00_SENS, SWC_CMD_SMR_CON,  TRUE, 1,{&nOTGT.mOut[3]}}, //PE1 Out1
		{4 ,&nINGT.mIn[3], STL_TM00_SENS, SWC_CMD_SMR_CON,  TRUE, 1,{&nOTGT.mOut[4]}}, //TE1
		{5 ,&nINGT.mIn[4], STL_TM00_SENS, SWC_CMD_SMR_CON,  TRUE, 1,{&nOTGT.mOut[5]}}, //TE2
		{6 ,&nINGT.mIn[5], STL_TM00_SENS, SWC_CMD_IDL_CON,  TRUE, 1,{&nOutGateDF}},    //TE3
		{7 ,&nINGT.mIn[6], STL_TM00_SENS, SWC_CMD_SMR_CON,  TRUE, 1,{&nOTGT.mOut[6]}}, //TE4
		{8 ,&nINGT.mIn[7], STL_TM00_SENS, SWC_CMD_SMR_CON,  TRUE, 1,{&nOTGT.mOut[7]}}, //TE5
		{9 ,&nINGT.mIn[8], STL_TM00_SENS, SWC_CMD_SMR_CON,  TRUE, 1,{&nOTGT.mOut[8]}}, //TE6
		{10,&nINGT.mIn[9], STL_TM00_SENS, SWC_CMD_SMR_CON,  TRUE, 1,{&nOTGT.mOut[9]}}, //TE7
	  }
	},
	//Switching For Direction 1
 }
};
#elif MYSYSTEM_ID == 1
SINPUTGATE nINGT = {10,{
{492,100, 0,  95,  20,  70,  30, 70, 1.0,2.0,20000.0 ,1.0,1.0,1000.0 ,550.0 ,0,0,0,0, BASE_GTE,MAX_GTE,0,SL02,PN00,SNS_SMART,P_LEVEL,ST_OPEN,ST_OPEN,SNS_MD_AUTO},
{492,100, 0,  95,  20,  70,  30, 70, 1.0,2.0,20000.0 ,1.0,1.0,1000.0 ,550.0 ,0,0,0,0, BASE_GTE,MAX_GTE,1,SL02,PN01,SNS_SMART,P_LEVEL,ST_OPEN,ST_INIT,SNS_MD_AUTO},
{489, 60, 0,  28,  20,  22,  21, 22, 0.0,3.0,250000.0,1.0,1.0,20400.0,600.0 ,0,0,0,0, BASE_GTE,MAX_GTE,2,SL02,PN02,SNS_SMART,P_PRESS,ST_OPEN,ST_OPEN,SNS_MD_AUTO},
{489,200, 0, 155, 145, 150, 145,150, 0.0,1.9,90000.0 ,1.0,1.0,1000.0 ,500.0 ,0,0,0,0, BASE_GTE,MAX_GTE,3,SL02,PN03,SNS_SMART,P_TEMPR,ST_OPEN,ST_OPEN,SNS_MD_AUTO},
{489,200, 0, 155, 145, 150, 145,150, 1.0,1.0,45000.0 ,1.0,1.0,1000.0 ,550.0 ,0,0,0,0, BASE_GTE,MAX_GTE,4,SL02,PN04,SNS_SMART,P_TEMPR,ST_OPEN,ST_OPEN,SNS_MD_AUTO},
{492,200, 0, 195, 185, 190, 185,190, 1.0,1.0,45000.0 ,1.0,1.0,1000.0 ,550.0 ,0,0,0,0, BASE_GTE,MAX_GTE,5,SL02,PN05,SNS_IDLES,P_TEMPR,ST_OPEN,ST_OPEN,SNS_MD_AUTO},
{492,200, 0, 195, 185, 190, 185,190, 0.0,1.0,90000.0 ,1.0,1.0,1000.0 ,500.0 ,0,0,0,0, BASE_GTE,MAX_GTE,6,SL02,PN06,SNS_SMART,P_TEMPR,ST_OPEN,ST_OPEN,SNS_MD_AUTO},
{492,200, 0, 195, 185, 190, 185,190, 1.0,1.0,45000.0 ,1.0,1.0,1000.0 ,550.0 ,0,0,0,0, BASE_GTE,MAX_GTE,7,SL02,PN07,SNS_SMART,P_TEMPR,ST_OPEN,ST_OPEN,SNS_MD_AUTO},
{489,200, 0, 155, 145, 150, 145,150, 1.0,1.0,45000.0 ,1.0,1.0,1000.0 ,550.0 ,0,0,0,0, BASE_GTE,MAX_GTE,8,SL03,PN00,SNS_SMART,P_TEMPR,ST_OPEN,ST_OPEN,SNS_MD_AUTO},
{492,200, 0, 195, 185, 190, 185,190, 1.0,1.0,45000.0 ,1.0,1.0,1000.0 ,550.0 ,0,0,0,0, BASE_GTE,MAX_GTE,9,SL03,PN01,SNS_SMART,P_TEMPR,ST_OPEN,ST_OPEN,SNS_MD_AUTO},
}};
SOUTPUTGATE nOTGT = {10,{
{0,5100,10,30,0.0,0.4,NZ,SDIR,0,SMART_GTE,SL04,PN02,"п.812/1"},//Lev LE1 RP4
{0,5100,15,30,0.0,0.4,NZ,SINV,0,SMART_GTE,SL04,PN03,"п.812/2"},//Lev LE1 RP3
{0,5100,20,30,0.2,1.0,NO,SDIR,0,SMART_GTE,SL04,PN00,"п.811/1"},//Prs PE1 RP2
{0,5100,25,30,0.2,0.8,NZ,SINV,0,SMART_GTE,SL04,PN01,"п.811/2"},//Prs PE1 RP1
{0,5100,30,30,0.2,1.0,NZ,SDIR,0,IDLES_GTE,SL04,PN05,"п.814"},  //Tmp TE1 RP5
{0,5100,35,30,0.2,1.0,NZ,SINV,0,IDLES_GTE,SL04,PN04,"п.815"},  //Tmp TE2 RP6
{0,5100,40,30,0.2,1.0,NZ,SDIR,0,IDLES_GTE,SL04,PN06,"п.813"},  //Tmp TE4 RP8
{0,5100,45,30,0.0,1.0,NO,SDIR,0,IDLES_GTE,SL05,PN00,"п.854"},  //Tmp TE5 RP10
{0,5100,50,30,0.0,1.0,NO,SDIR,0,IDLES_GTE,SL05,PN01,"п.855"},  //Tmp TE6 RP9
{0,5100,55,30,0.2,1.0,NZ,SDIR,0,IDLES_GTE,SL04,PN07,"п.511"},  //Tmp TE7 RP7
}};
SSOFTSWITCHTABLE  nSoftSwitchTable=
{
 0,"Switching Table For System AC-2",1,
 {
	//Switching For Direction 0
	{
      0,1,11,&nINGT,&nOTGT,
	  {//ID  In_Gate     Conn Type     AmOut  Out_Gate_0  Out_Gate_1
		{0 ,&nINGT.mIn[0], STL_LV00_SENS, SWC_CMD_SMR_CON, TRUE, 1,{&nOTGT.mOut[0]}},//LE
		{1 ,&nINGT.mIn[0], STL_LV00_SENS, SWC_CMD_SMR_CON, TRUE, 1,{&nOTGT.mOut[1]}},//LE
		{2 ,&nINGT.mIn[2], STL_PS00_SENS, SWC_CMD_SMR_CON, TRUE, 1,{&nOTGT.mOut[2]}},//PE
		{3 ,&nINGT.mIn[2], STL_PS00_SENS, SWC_CMD_SMR_CON, TRUE, 1,{&nOTGT.mOut[3]}},//PE
		{4 ,&nINGT.mIn[3], STL_TM00_SENS, SWC_CMD_SMR_CON, TRUE, 1,{&nOTGT.mOut[4]}},//TE1
		{5 ,&nINGT.mIn[4], STL_TM00_SENS, SWC_CMD_SMR_CON, TRUE, 1,{&nOTGT.mOut[5]}},//TE2
		{6 ,&nINGT.mIn[5], STL_TM00_SENS, SWC_CMD_IDL_CON, TRUE, 1,{&nOutGateDF}},   //TE3
		{7 ,&nINGT.mIn[6], STL_TM00_SENS, SWC_CMD_SMR_CON, TRUE, 1,{&nOTGT.mOut[6]}},//TE4
		{8 ,&nINGT.mIn[7], STL_TM00_SENS, SWC_CMD_SMR_CON, TRUE, 1,{&nOTGT.mOut[7]}},//TE5
		{9 ,&nINGT.mIn[8], STL_TM00_SENS, SWC_CMD_SMR_CON, TRUE, 1,{&nOTGT.mOut[8]}},//TE6
		{10,&nINGT.mIn[9], STL_TM00_SENS, SWC_CMD_SMR_CON, TRUE, 1,{&nOTGT.mOut[9]}},//TE7
	  }
	},
	//Switching For Direction 1
 }
};
#elif MYSYSTEM_ID == 2
SINPUTGATE nINGT = {11,{
{492,100, 0,  95,  20,  70,  30, 60, 1.0,2.0,20000.0 ,1.0,1.0,1000.0 ,550.0 ,0,0,0,0, BASE_GTE,MAX_GTE, 0,SL02,PN00,SNS_SMART,P_LEVEL,ST_OPEN,ST_OPEN,SNS_MD_AUTO},
{492,100, 0,  95,  20,  70,  30, 65, 1.0,2.0,20000.0 ,1.0,1.0,1000.0 ,550.0 ,0,0,0,0, BASE_GTE,MAX_GTE, 1,SL02,PN01,SNS_SMART,P_LEVEL,ST_OPEN,ST_OPEN,SNS_MD_AUTO},
{492,100, 0,  95,  20,  70,  30, 70, 1.0,2.0,20000.0 ,1.0,1.0,1000.0 ,550.0 ,0,0,0,0, BASE_GTE,MAX_GTE, 2,SL02,PN02,SNS_SMART,P_LEVEL,ST_OPEN,ST_OPEN,SNS_MD_AUTO},
{489, 60, 0,  28,  20,  22,  21, 22, 0.0,3.0,250000.0,1.0,1.0,20400.0,600.0 ,0,0,0,0, BASE_GTE,MAX_GTE, 3,SL02,PN03,SNS_SMART,P_PRESS,ST_OPEN,ST_OPEN,SNS_MD_AUTO},
{489,200, 0, 155, 145, 150, 145,150, 0.0,1.9,90000.0 ,1.0,1.0,1000.0 ,500.0 ,0,0,0,0, BASE_GTE,MAX_GTE, 4,SL02,PN04,SNS_SMART,P_TEMPR,ST_OPEN,ST_OPEN,SNS_MD_AUTO},
{489,200, 0, 155, 145, 150, 145,150, 1.0,1.0,45000.0 ,1.0,1.0,1000.0 ,550.0 ,0,0,0,0, BASE_GTE,MAX_GTE, 5,SL02,PN05,SNS_SMART,P_TEMPR,ST_OPEN,ST_OPEN,SNS_MD_AUTO},
{492,200, 0, 195, 185, 190, 185,190, 1.0,1.0,45000.0 ,1.0,1.0,1000.0 ,550.0 ,0,0,0,0, BASE_GTE,MAX_GTE, 6,SL02,PN06,SNS_IDLES,P_TEMPR,ST_OPEN,ST_OPEN,SNS_MD_AUTO},
{492,200, 0, 195, 185, 190, 185,190, 0.0,1.0,90000.0 ,1.0,1.0,1000.0 ,500.0 ,0,0,0,0, BASE_GTE,MAX_GTE, 7,SL02,PN07,SNS_SMART,P_TEMPR,ST_OPEN,ST_OPEN,SNS_MD_AUTO},
{492,200, 0, 195, 185, 190, 185,190, 1.0,1.0,45000.0 ,1.0,1.0,1000.0 ,550.0 ,0,0,0,0, BASE_GTE,MAX_GTE, 8,SL03,PN00,SNS_SMART,P_TEMPR,ST_OPEN,ST_OPEN,SNS_MD_AUTO},
{489,200, 0, 155, 145, 150, 145,150, 1.0,1.0,45000.0 ,1.0,1.0,1000.0 ,550.0 ,0,0,0,0, BASE_GTE,MAX_GTE, 9,SL03,PN01,SNS_SMART,P_TEMPR,ST_OPEN,ST_OPEN,SNS_MD_AUTO},
{492,200, 0, 195, 185, 190, 185,190, 1.0,1.0,45000.0 ,1.0,1.0,1000.0 ,550.0 ,0,0,0,0, BASE_GTE,MAX_GTE,10,SL03,PN02,SNS_SMART,P_TEMPR,ST_OPEN,ST_OPEN,SNS_MD_AUTO},
}};
SOUTPUTGATE nOTGT = {10,{
{0,5100,10,30,0.0,0.4,NZ,SDIR,0,SMART_GTE,SL04,PN02,"п.812/1"},//Lev LE1 RP4
{0,5100,15,30,0.0,0.4,NZ,SINV,0,SMART_GTE,SL04,PN03,"п.812/2"},//Lev LE1 RP3
{0,5100,20,30,0.2,1.0,NO,SDIR,0,SMART_GTE,SL04,PN00,"п.811/1"},//Prs PE1 RP2
{0,5100,25,30,0.2,0.8,NZ,SINV,0,SMART_GTE,SL04,PN01,"п.811/2"},//Prs PE1 RP1
{0,5100,30,30,0.2,1.0,NZ,SDIR,0,IDLES_GTE,SL04,PN05,"п.814"},  //Tmp TE1 RP5
{0,5100,35,30,0.2,1.0,NZ,SINV,0,IDLES_GTE,SL04,PN04,"п.815"},  //Tmp TE2 RP6
{0,5100,40,30,0.2,1.0,NZ,SDIR,0,IDLES_GTE,SL04,PN06,"п.813"},  //Tmp TE4 RP8
{0,5100,45,30,0.0,1.0,NO,SDIR,0,IDLES_GTE,SL05,PN00,"п.854"},  //Tmp TE5 RP10
{0,5100,50,30,0.0,1.0,NO,SDIR,0,IDLES_GTE,SL05,PN01,"п.855"},  //Tmp TE6 RP9
{0,5100,55,30,0.2,1.0,NZ,SDIR,0,IDLES_GTE,SL04,PN07,"п.511"},  //Tmp TE7 RP7
}};
SSOFTSWITCHTABLE  nSoftSwitchTable=
{
 0,"Switching Table For System AC-3",1,
 {
	//Switching For Direction 0
	{
      0,2,11,&nINGT,&nOTGT,
	  {//ID   SL   PN        Conn Type AmOut  Out_Gate_0  Out_Gate_1      SParam
		{0 ,&nINGT.mIn[1], STL_LV00_SENS, SWC_CMD_SMR_CON, TRUE, 1,{&nOTGT.mOut[0]}},
		{1 ,&nINGT.mIn[1], STL_LV00_SENS, SWC_CMD_SMR_CON, TRUE, 1,{&nOTGT.mOut[1]}},
		{2 ,&nINGT.mIn[3], STL_PS00_SENS, SWC_CMD_SMR_CON, TRUE, 1,{&nOTGT.mOut[2]}},
		{3 ,&nINGT.mIn[3], STL_PS00_SENS, SWC_CMD_SMR_CON, TRUE, 1,{&nOTGT.mOut[3]}},
		{4 ,&nINGT.mIn[4], STL_TM00_SENS, SWC_CMD_SMR_CON, TRUE, 1,{&nOTGT.mOut[4]}},
		{5 ,&nINGT.mIn[5], STL_TM00_SENS, SWC_CMD_SMR_CON, TRUE, 1,{&nOTGT.mOut[5]}},
		{6 ,&nINGT.mIn[6], STL_TM00_SENS, SWC_CMD_IDL_CON, TRUE, 1,{&nOutGateDF}},
		{7 ,&nINGT.mIn[7], STL_TM00_SENS, SWC_CMD_SMR_CON, TRUE, 1,{&nOTGT.mOut[6]}},
		{8 ,&nINGT.mIn[8], STL_TM00_SENS, SWC_CMD_SMR_CON, TRUE, 1,{&nOTGT.mOut[7]}},
		{9 ,&nINGT.mIn[9], STL_TM00_SENS, SWC_CMD_SMR_CON, TRUE, 1,{&nOTGT.mOut[8]}},
		{10,&nINGT.mIn[10], STL_TM00_SENS, SWC_CMD_SMR_CON, TRUE, 1,{&nOTGT.mOut[9]}},
	  }
	},
	//Switching For Direction 1
 }
};
#elif MYSYSTEM_ID == 3

SINPUTGATE nINGT = {12,{
{492,100, 0,  95,  20,  70,  30, 60, 1.0,2.0,20000.0 ,1.0,1.0,1000.0 ,550.0 ,0,0,0,0, BASE_GTE,MAX_GTE, 0,SL02,PN00,SNS_SMART,P_LEVEL,ST_OPEN,ST_OPEN,SNS_MD_AUTO},
{492,100, 0,  95,  20,  70,  30, 65, 1.0,2.0,20000.0 ,1.0,1.0,1000.0 ,550.0 ,0,0,0,0, BASE_GTE,MAX_GTE, 1,SL02,PN01,SNS_SMART,P_LEVEL,ST_OPEN,ST_OPEN,SNS_MD_AUTO},
{492,100, 0,  95,  20,  70,  30, 70, 1.0,2.0,20000.0 ,1.0,1.0,1000.0 ,550.0 ,0,0,0,0, BASE_GTE,MAX_GTE, 2,SL02,PN02,SNS_SMART,P_LEVEL,ST_OPEN,ST_OPEN,SNS_MD_AUTO},
{492,100, 0,  95,  20,  70,  30, 70, 1.0,2.0,20000.0 ,1.0,1.0,1000.0 ,550.0 ,0,0,0,0, BASE_GTE,MAX_GTE, 3,SL02,PN03,SNS_SMART,P_LEVEL,ST_OPEN,ST_OPEN,SNS_MD_AUTO},
{492,100, 0,  95,  20,  70,  30, 70, 1.0,2.0,20000.0 ,1.0,1.0,1000.0 ,550.0 ,0,0,0,0, BASE_GTE,MAX_GTE, 4,SL02,PN04,SNS_SMART,P_LEVEL,ST_OPEN,ST_OPEN,SNS_MD_AUTO},
{492,100, 0,  95,  20,  70,  30, 70, 1.0,2.0,20000.0 ,1.0,1.0,1000.0 ,550.0 ,0,0,0,0, BASE_GTE,MAX_GTE, 5,SL02,PN05,SNS_SMART,P_LEVEL,ST_OPEN,ST_OPEN,SNS_MD_AUTO},
{492,100, 0,  95,  20,  70,  30, 70, 1.0,2.0,20000.0 ,1.0,1.0,1000.0 ,550.0 ,0,0,0,0, BASE_GTE,MAX_GTE, 6,SL02,PN06,SNS_SMART,P_LEVEL,ST_OPEN,ST_OPEN,SNS_MD_AUTO},
{492,100, 0,  95,  20,  70,  30, 70, 1.0,2.0,20000.0 ,1.0,1.0,1000.0 ,550.0 ,0,0,0,0, BASE_GTE,MAX_GTE, 7,SL02,PN07,SNS_SMART,P_LEVEL,ST_OPEN,ST_OPEN,SNS_MD_AUTO},
{492, 60, 0,  28,   2,  22,  3,  10, 0.0,3.0,250000.0,1.0,1.0,20400.0,600.0 ,0,0,0,0, BASE_GTE,MAX_GTE, 8,SL03,PN00,SNS_SMART,P_PRESS,ST_OPEN,ST_OPEN,SNS_MD_AUTO},
{492, 60, 0,  28,   2,  22,  3,  10, 0.0,3.0,250000.0,1.0,1.0,20400.0,600.0 ,0,0,0,0, BASE_GTE,MAX_GTE, 9,SL03,PN01,SNS_SMART,P_PRESS,ST_OPEN,ST_OPEN,SNS_MD_AUTO},
{492,200, 0, 160,  30, 150,  40, 50, 0.0,1.9,90000.0 ,1.0,1.0,1000.0 ,500.0 ,0,0,0,0, BASE_GTE,MAX_GTE,10,SL03,PN02,SNS_IDLES,P_TEMPR,ST_OPEN,ST_OPEN,SNS_MD_AUTO},
{492,200, 0, 160,  30, 150,  40, 50, 0.0,1.9,90000.0 ,1.0,1.0,1000.0 ,500.0 ,0,0,0,0, BASE_GTE,MAX_GTE,11,SL03,PN03,SNS_SMART,P_TEMPR,ST_OPEN,ST_OPEN,SNS_MD_AUTO},
}};
SOUTPUTGATE nOTGT = {7,{
{0,5100,10,30,0.2,1.0,NZ,SDIR,0,SMART_GTE,SL04,PN03,"п.820/1"},
{0,5100,15,30,0.2,1.0,NZ,SINV,0,SMART_GTE,SL04,PN04,"п.820/2"},
{0,5100,20,30,0.2,1.0,NZ,SDIR,0,SMART_GTE,SL04,PN00,"п.835/1"},
{0,5100,25,30,0.2,1.0,NZ,SDIR,0,SMART_GTE,SL04,PN01,"п.810/1"},
{0,5100,30,30,0.2,1.0,NO,SDIR,0,SMART_GTE,SL04,PN02,"п.822/1"},
{0,5100,35,30,0.2,1.0,NZ,SDIR,0,SMART_GTE,SL04,PN05,"п.841/1"},
{0,5100,40,30,0.2,1.0,NO,SDIR,0,SMART_GTE,SL04,PN06,"п.841/2"},
}};

SSOFTSWITCHTABLE  nSoftSwitchTable=
{
 0,"Switching Table For System #4",1,
 {
	//Switching For Direction 0
	{
      0,3,8,&nINGT,&nOTGT,
	  {     //Type     Slot PinN   Switch Command    Slot PinN Sens Info
		{0,&nINGT.mIn[0], STL_LVN4_SENS, SWC_CMD_SMR_CON,  TRUE, 1,{&nOTGT.mOut[5]}},
		{1,&nINGT.mIn[2], STL_LVN4_SENS, SWC_CMD_SMR_CON,  TRUE, 1,{&nOTGT.mOut[6]}},
		{2,&nINGT.mIn[4], STL_LV04_SENS, SWC_CMD_SMR_CON,  TRUE, 1,{&nOTGT.mOut[0]}},
		{3,&nINGT.mIn[4], STL_LV04_SENS, SWC_CMD_SMR_CON,  TRUE, 1,{&nOTGT.mOut[1]}},
		{4,&nINGT.mIn[8], STL_PS04_SENS, SWC_CMD_SMR_CON,  TRUE, 1,{&nOTGT.mOut[2]}},
		{5,&nINGT.mIn[9], STL_PS04_SENS, SWC_CMD_SMR_CON,  TRUE, 1,{&nOTGT.mOut[3]}},
		{6,&nINGT.mIn[10],STL_TM00_SENS, SWC_CMD_IDL_CON,  TRUE, 1,{&nOutGateDF}},
		{7,&nINGT.mIn[11],STL_TM00_SENS, SWC_CMD_SMR_CON,  TRUE, 1,{&nOTGT.mOut[4]}},
	  }
	},
 }
};
#elif MYSYSTEM_ID == 4
SDIGGATES nINGT = {10,{
{8,  {{02,00},{02,01},{02,02},{02,03}, {03, 7},{03, 9},{03,10},{03,11}}}, //DI_02
{8,  {{02, 4},{02, 5},{02, 6},{02, 7}, {03,12},{03,13},{03,14},{03,15}}}, //DI_02
{8,  {{02, 8},{02, 9},{02,10},{02,11}, {03,16},{03,17},{03,18},{03,19}}}, //DI_02
{8,  {{02,12},{02,13},{02,14},{02,15}, {03,20},{03,21},{03,22},{03,23}}}, //DI_02
{8,  {{02,16},{02,17},{02,18},{02,19}, {03,24},{03,25},{03,26},{03,27}}}, //DI_03
{8,  {{02,20},{02,21},{02,22},{02,23}, {03,28},{03,29},{03,30},{03,31}}}, //DI_03
{8,  {{02,24},{02,25},{02,26},{02,27},{02,28},{02,29},{02,30},{02,31}}}, //DI_03
{8,  {{03,00},{03,01},{03,02},{03,03},{03,04},{03,05},{03,06},{03, 8}}}, //DI_03
{16, {{04,00},{04,01},{04,02},{04,03},{04,04},{04,05},{04,06},{04,07},{04, 8},{04, 9},{04,10},{04,11},{04,12},{04,13},{04,14},{04,15}}},//DI_04
{16, {{04,16},{02,17},{04,18},{04,19},{04,20},{04,21},{04,22},{04,23},{04,24},{04,25},{04,26},{04,27},{04,28},{04,29},{04,30},{04,31}}},//DI_04
}};
SDIGGATES nOTGT = {10,{
{4, {{07,01},{07,00},{05,01},{05,00}}}, //DO_05 1
{4, {{07,02},{07,03},{05,02},{05,03}}}, //DO_05 2
{4, {{07,05},{07,04},{05,05},{05,04}}}, //DO_06 3
{4, {{07,06},{07,07},{05,06},{05,07}}}, //DO_06 4
{4, {{ 8,01},{ 8,00},{06,01},{06,00}}}, //DO_07 5
{4, {{ 8,02},{ 8,03},{06,02},{06,03}}}, //DO_07 6
{4, {{ 8,05},{ 8,04},{06,05},{06,04}}}, //DO_08 7
{4, {{ 8,06},{ 8,07},{06,06},{06,07}}}, //DO_08 8
{8, {{ 9,00},{ 9,01},{ 9,02},{ 9,03},{ 9,04},{ 9,05},{ 9,06},{ 9,07}}}, //DO_09
{8, {{10,00},{10,01},{10,02},{10,03},{10,04},{10,05},{10,06},{10,07}}}, //DO_10
}};
//Input Gate Section (Model 20in X 8out)
SSOFTSWITCHTABLE  nSoftSwitchTable=
{
 0,"Switching Table For System #5",1,
 {
	//Switching For Direction 0
	{
      0,4,10,&nINGT,&nOTGT,
	  {     //Type     Slot PinN   Switch Command    Slot PinN Sens Info
		{0 ,&nINGT.sIoGate[0], STL_DIGS00_SENS, SWC_CMD_LOG_CON, TRUE, 1,{&nOTGT.sIoGate[0]}},
		{1 ,&nINGT.sIoGate[3], STL_DIGS00_SENS, SWC_CMD_LOG_CON, TRUE, 1,{&nOTGT.sIoGate[3]}},
		{2 ,&nINGT.sIoGate[1], STL_DIGS00_SENS, SWC_CMD_LOG_CON, TRUE, 1,{&nOTGT.sIoGate[1]}},
		{3 ,&nINGT.sIoGate[4], STL_DIGS00_SENS, SWC_CMD_LOG_CON, TRUE, 1,{&nOTGT.sIoGate[4]}},
		{4 ,&nINGT.sIoGate[2], STL_DIGS00_SENS, SWC_CMD_LOG_CON, TRUE, 1,{&nOTGT.sIoGate[2]}},
		{5 ,&nINGT.sIoGate[5], STL_DIGS00_SENS, SWC_CMD_LOG_CON, TRUE, 1,{&nOTGT.sIoGate[5]}},
		{6 ,&nINGT.sIoGate[6], STL_DIGS00_SENS, SWC_CMD_LOG_CON, TRUE, 1,{&nOTGT.sIoGate[6]}},
		{7 ,&nINGT.sIoGate[7], STL_DIGS00_SENS, SWC_CMD_LOG_CON, TRUE, 1,{&nOTGT.sIoGate[7]}},
		{8 ,&nINGT.sIoGate[8], STL_DIGS00_SENS, SWC_CMD_LOG_CON, TRUE, 1,{&nOTGT.sIoGate[8]}},
		{9 ,&nINGT.sIoGate[9], STL_DIGS00_SENS, SWC_CMD_LOG_CON, TRUE, 1,{&nOTGT.sIoGate[9]}},
	  }
	},
 }
};
#elif MYSYSTEM_ID == 5
/*
//Датчик давления
typedef struct _tagTPRParam
{
	BYTE byID;
	BYTE byAmParam;
	BYTE byType;
	BYTE bySlot;
	BYTE byPin;
	BYTE byAlmState;
	BYTE byState;
	WORD wJob;
	WORD wParam;
}STPRPARAM;
*/
STPRPARAMS nTPR = {2,TPR,{
{0  ,0  ,TPR ,4, 0, EN_OPEN, PRI_HI, 10, 5},
{1  ,1  ,TPR ,4, 1, EN_OPEN, PRI_HI, 11, 7},
}};
/*
//Датчик температуры
typedef struct _tagTTMParam
{
	BYTE byID;
	BYTE byAmParam;
	BYTE byType;
	BYTE bySlot;
	BYTE byPin;
	BYTE byAlmState;
	BYTE byState;
	WORD wJob;
	WORD wParam;
}STTMPARAM;
*/
STTMPARAMS nTTM = {2,TTM,{
{2  ,0  ,TTM ,5, 0, EN_OPEN, PRI_HI, 30, 20},
{3  ,1  ,TTM ,5, 1, EN_OPEN, PRI_HI, 25, 20},
}};
/*
//Счетчики импульсов
typedef struct _tagTCParam
{
	BYTE byID;
	BYTE byAmParam;
	BYTE byType;
	BYTE bySlot;
	BYTE byPin;
	BYTE byAlmState;
	BYTE byState;
	FLOAT fKoeff;
	DWORD dwMaxFreq;
	DWORD dwParam;
}STCPARAM;
*/
STCPARAMS nTC = {16,TC,{
{4  ,0  ,TC ,0, 0, EN_OPEN, PRI_HI, 10000,1.23, 11},
{5  ,1  ,TC ,0, 0, EN_OPEN, PRI_HI, 10000,2.45, 21},
{6  ,2  ,TC ,0, 0, EN_OPEN, PRI_HI, 10000,3.23, 31},
{7  ,3  ,TC ,0, 0, EN_OPEN, PRI_HI, 10000,4.23, 41},

{8  ,4  ,TC ,0, 0, EN_OPEN, PRI_HI, 1000 ,5.234, 51},
{9  ,5  ,TC ,0, 0, EN_OPEN, PRI_HI, 1000 ,6.456, 61},
{10 ,6  ,TC ,0, 0, EN_OPEN, PRI_HI, 1000 ,7.23, 71},
{11 ,7  ,TC ,0, 0, EN_OPEN, PRI_HI, 1000 ,8.345, 81},

{12 ,8  ,TC ,0, 0, EN_OPEN, PRI_HI, 1000 ,9.234, 91},
{13 ,9  ,TC ,0, 0, EN_OPEN, PRI_HI, 1000 ,10.234,101},
{14 ,10 ,TC ,0, 0, EN_OPEN, PRI_HI, 1000 ,11.23,111},
{15 ,11 ,TC ,0, 0, EN_OPEN, PRI_HI, 1000 ,12.234,121},

{16 ,12 ,TC ,0, 0, EN_OPEN, PRI_HI, 1000 ,0.345,131112},
{17 ,13 ,TC ,0, 0, EN_OPEN, PRI_HI, 1000 ,0.145,141112},
{18 ,14 ,TC ,0, 0, EN_OPEN, PRI_HI, 1000 ,0.235,151112},
{19 ,15 ,TC ,0, 0, EN_OPEN, PRI_HI, 1000 ,0.134,161112},
}};
/*
//Частотный привод
typedef struct _tagTFParam
{
BYTE byID;
BYTE byAmParam;
BYTE byType;
BYTE bySlot; //Для задания
BYTE byPin;  //Для задания

BYTE bySlot1; //Запуск
BYTE byPin1;  //Запуск

BYTE bySlot2; //Останов
BYTE byPin2;  //Останов

BYTE bySlot3; //Авария1
BYTE byPin3;  //Авария1

BYTE bySlot4; //Авария2
BYTE byPin4;  //Авария2

BYTE byStartST;
BYTE byStopST;
BYTE byAlST0;
BYTE byAlST1;
WORD wTask;
WORD wParam;
}STFPARAM;
*/
STFPARAMS nTF = {3,TF,{
{20 ,0  ,TF ,6, 0, 9, 0, 9, 1, 7, 0, 7, 1, 0, 50, 30},
{21 ,1  ,TF ,6, 1, 9, 2, 9, 3, 7, 2, 7, 3, 0, 60, 20},
{22 ,1  ,TF ,6, 1, 9, 4, 9, 5, 7, 4, 7, 5, 0, 65, 10},
}};
/*
//Управляемые краны
typedef struct _tagTKParam
{
BYTE byID;
BYTE byAmParam;
BYTE byType;
BYTE bySlot;  //Запуск
BYTE byPin;   //Запуск
BYTE bySlot1; //Останов
BYTE byPin1;  //Останов
BYTE byStOP;
BYTE byStCL;
BYTE byStMD;
WORD wMaxOpenTime;
REAL fJobOpen;
REAL fOpenState;
}STKPARAM;
*/
STKPARAMS nTKP = {4,TKP,{
{23  ,0  ,TKP,10,0 ,10, 1, 0,0,0, 40,0,0},
{24  ,1  ,TKP,10,2 ,10, 3, 0,0,0, 40,0,0},
{25  ,2  ,TKP,10,4 ,10, 5, 0,0,0, 40,0,0},
{26  ,3  ,TKP,10,6 ,10, 7, 0,0,0, 40,0,0},
}};
/*
//Перекидное устройство
typedef struct _tagPUParam
{
BYTE byID;
BYTE byAmParam;
BYTE byType;
BYTE bySlot;
BYTE byPin;
BYTE bySlot1;
BYTE byPin1;
BYTE bySlot2;
BYTE byPin2;
BYTE bySlot3;
BYTE byPin3;
WORD wSt0;
DWORD dwMaxTime;
DWORD dwOpenTime;
}SPUPARAM;
*/
SPUPARAMS nTPU = {2,TPU,{
{27  ,0  ,TPU ,9 ,6 ,7 ,8 ,7 ,9 ,7 ,10, 0, 40, 0},
{28  ,1  ,TPU ,9 ,7 ,7 ,11,8 ,0 ,8 ,1 , 0, 40, 0},
}};
/*
typedef struct _tagTSParam
{
    BYTE byID;
    BYTE byAmParam;
	BYTE byType;
	BYTE bySlot;
	BYTE byPin;
	BYTE byState;
	BYTE byCRemPulce;
	BYTE byCSetPulce;
	BYTE byAlarmMode;
	BYTE byPriority;
	BYTE byParam;
}STSPARAM;
*/
STSMPARAMS nTS = {8,TS,{
{29  ,0 ,TS ,8 ,4 , 0, EN_OPEN, PRI_HI, 5, 5, EN_AL_TO_AL, 0},
{30  ,1 ,TS ,8 ,5 , 0, EN_OPEN, PRI_HI, 5, 5, EN_AL_TO_AL, 0},
{31  ,2 ,TS ,8 ,6 , 0, EN_OPEN, PRI_HI, 5, 5, EN_AL_TO_AL, 0},
{32  ,3 ,TS ,8 ,7 , 0, EN_OPEN, PRI_HI, 5, 5, EN_AL_TO_AL, 0},
{33  ,4 ,TS ,8 ,8 , 0, EN_OPEN, PRI_HI, 5, 5, EN_AL_TO_AL, 0},
{34  ,5 ,TS ,8 ,9 , 0, EN_OPEN, PRI_HI, 5, 5, EN_AL_TO_AL, 0},
{35  ,6 ,TS ,8 ,10, 0, EN_OPEN, PRI_HI, 5, 5, EN_AL_TO_AL, 0},
{36  ,7 ,TS ,8 ,11, 0, EN_OPEN, PRI_HI, 5, 5, EN_AL_TO_AL, 0},
}};
/*
typedef struct _tagTUParam
{
	BYTE byID;
	BYTE byAmParam;
	BYTE byType;
	BYTE bySlot;
	BYTE byPin;
	BYTE byAlmState;
	BYTE byState;
	BYTE byPulceType;
    BYTE byCSetPulce;
	BYTE byParam;
}STUPARAM;
*/
STUMPARAMS nTU = {8,TU,{
{37  ,0 ,TU ,9 ,8 , 0, EN_OPEN, EN_DIRECT, 10, 0},
{38  ,1 ,TU ,9 ,9 , 0, EN_OPEN, EN_DIRECT, 10, 0},
{39  ,2 ,TU ,9 ,10, 0, EN_OPEN, EN_DIRECT, 10, 0},
{40  ,3 ,TU ,9 ,11, 0, EN_OPEN, EN_DIRECT, 20, 0},
{41  ,4 ,TU ,10,8 , 0, EN_OPEN, EN_DIRECT, 20, 0},
{42  ,5 ,TU ,10,9 , 0, EN_OPEN, EN_DIRECT, 30, 0},
{43  ,6 ,TU ,10,10, 0, EN_OPEN, EN_DIRECT, 40, 0},
{44  ,7 ,TU ,10,11, 0, EN_OPEN, EN_DIRECT, 50, 0},
}};
/*
typedef struct _tagTVSParam
{
BYTE byID;
BYTE byAmParam;
BYTE byType;
STVSDATA sDT;
}STVSPARAM;
0000.00000
0001.00000
*/
STVSPARAMS nTVS = {2,TVS,{
{45  ,0  ,TVS ,0x01,0x02,0x01,0x01,0x01,0x01,0x01,0x01,0x01,0x01,0x01},
{46  ,1  ,TVS ,0x30,0x30,0x30,0x31,0x2e,0x30,0x31,0x32,0x33,0x34,0x05},
}};
//Измеритель уровня
/*
typedef struct _tagLVParam
{
	BYTE byID;
	BYTE byAmParam;
	BYTE byType;
	BYTE bySlot;
	BYTE byPin;
	BYTE bySlot1;
	BYTE byPin1;
    SLVDATA sDT;
}SLVPARAM;
*/
SLVPARAMS nLV = {1,TLV,{
{47  ,0  ,TLV,8 ,2 ,8 ,3,0,95,75,0},
}};
/*
//Модуль слежения
typedef struct _tagODSData
{
	//BYTE byAutoStart;
	//BYTE byPreStart;
	//BYTE byStart;
	//BYTE byStop;
	//BYTE byFinish;
    //BYTE byMode;
    DWORD dwSysState;
	WORD wJTMPreStart;
	WORD wTMPreStart;
	WORD wJTMStart;
	WORD wTMtart;
}SOBSMDATA;
*/
SOBSPARAMS nOS = {1,TOS,{
{48  ,0  ,TOS ,0, 0, EN_OPEN, PRI_HI, 0x00000000,10,0,30,0,20,0},
}};

STIPARAMS nTI = {2,TI,{
{42  ,0  ,TI ,2, 0, 0, EN_OPEN, PRI_HI, 5, 27000, 25000, 15000, 10000, 5000, 32760, 3000, 0},
{43  ,1  ,TI ,2, 1, 0, EN_OPEN, PRI_HI, 5, 29000, 28000, 19000, 18000, 5000, 32760, 3276, 0},
}};
/*
&nTPR,&nTTM,&nTC,&nTF,&nTKP,&nTPU,&nTS,&nTU,
*/
SSOFTSWITCHTABLE  nSoftSwitchTable=
{
 0,"Switching Table For System #5",1,
 {
	//Switching For Direction 0
	{
      0,1,11,49,0,0,0,NULL,NULL,
	  { //Type     Slot PinN   Switch Command    Slot PinN Sens Info
		//TI - AI Module
	    &nTPR,
		&nTTM,
		&nTC,
		&nTF,
		&nTKP,
		&nTPU,
		&nTS,
		&nTU,
		&nTVS,
		&nLV,
		&nOS,
		//&nPL,
		//&nTM,
		//&nTAL,
	  }
	},
 }
};
#endif
#ifdef WIN32
	int SYSxinfo(SYSxinfo_typ *p){return 0;};
#endif
```

#### bnrcyclicsystem.c
```c
/********************************************************************
 * COPYRIGHT -- Kontora
 ********************************************************************
 * Program: bnrmain
 * File: bnrlsens.c
 * Author: Abramenya
 * Created: January 19, 2009
 *******************************************************************/

#include "bnrcyclicsystem.h"
#ifdef _DEFAULT_INCLUDES
 #include <AsDefault.h>
#endif
SINT *chProcState[] =
{
	 "OFF",
 	 "ON"
};
DECLARE_TASKCHAIN(SkipCC)
{
    {EXIT_D}
};
DECLARE_STATE(BadStateCC)
{
    {EV_UNKNOWN_REQ, SkipCC}
};
DECLARE_STATELIST(StateListCC)
{
    {S_BAD, BadStateCC}
};
BOOL CCyclicSystem_SetState(This,TStateCode vNewState)
{
	 DECLARE_SINGLE_OPEN(CCyclicSystem)
     TStateList * pvList = pT->GetStateList(pC);
     pT->m_pvState = pvList[(INT16)vNewState].m_pvState;
     pT->m_vState  = vNewState;
	 //pT->v[STATE] = vNewState;
     return TRUE;
}
BOOL CCyclicSystem_HandleEvent(This,TEvent vEvent)
{
	 DECLARE_SINGLE_OPEN(CCyclicSystem)
	 TState* pvState;
     for(pvState=pT->m_pvState; pvState->m_vEvent!=EV_UNKNOWN_REQ; pvState++)
	 {
        if(pvState->m_vEvent==vEvent)
        {
            return pT->HandleTask(pC,pvState->m_pvTask);
        }
	 }
     return FALSE;
}
BOOL CCyclicSystem_HandleTask(This,TTask* pvTask)
{
	 DECLARE_SINGLE_OPEN(CCyclicSystem)
     return (*pvTask==EXIT_D)?TRUE:FALSE;
}
TStateList* CCyclicSystem_GetStateList(This)
{
	 DECLARE_SINGLE_OPEN(CCyclicSystem)
     return (TStateList*)&StateListCC;
}
TStateCode CCyclicSystem_GetStateCode(This)
{
	 DECLARE_SINGLE_OPEN(CCyclicSystem)
	 return pT->m_vState;
}
TState* CCyclicSystem_GetState(This)
{
	 DECLARE_SINGLE_OPEN(CCyclicSystem)
	 return pT->m_pvState;
}
void CCyclicSystem_SetMsgAuto(This,SMESSAGE *pMsg)
{
     DECLARE_SINGLE_OPEN(CCyclicSystem)
	 BYTE byEvent = pMsg->m_sbyType;
	 pT->HandleEvent(pT,byEvent);
}
void CCyclicSystem_SetAutoState(This,TStateCode vNewState)
{
     DECLARE_SINGLE_OPEN(CCyclicSystem)
	 pT->SetState(pT,vNewState);
}
/////////////////////////////////////////////////////////////////
void CCyclicSystem_Create(This,SINT* chProcName,BYTE byStateProc,BYTE byPeriod)
{
     //DECLARE_SINGLE_OPEN(CCyclicSystem)
	 DECLARE_SINGLE_OPEN(CCyclicSystem)
	 pT->SetName(pT,chProcName);
	 pT->SetStateProc(pT,byStateProc);
	 pT->SetPeriod(pT,byPeriod);
	 pT->m_dwAmoutQuant = 0;
	 #ifdef DEB_CCyclicSystem
	 Info("\n(__)CYCLS::>Create Process::State:%s Period:%b Process:%s.",chProcState[byStateProc],&byPeriod,chProcName);
     #endif
}
void CCyclicSystem_CreateSuspend(This,SINT* chProcName,BYTE byPeriod)
{
	 //DECLARE_SINGLE_OPEN(CCyclicSystem)
	 DECLARE_SINGLE_OPEN(CCyclicSystem)
	 pT->SetName(pT,chProcName);
	 pT->Stop(pT);
	 pT->SetPeriod(pT,byPeriod);
}
void CCyclicSystem_Start(This)
{
     //DECLARE_SINGLE_OPEN(CCyclicSystem)
	 DECLARE_SINGLE_OPEN(CCyclicSystem)
	 pT->SetStateProc(pT,DEV_CJOB_ST_RESM);
}
void CCyclicSystem_Stop(This)
{
     //DECLARE_SINGLE_OPEN(CCyclicSystem)
	 DECLARE_SINGLE_OPEN(CCyclicSystem)
	 pT->SetStateProc(pT,DEV_CJOB_ST_SUSP);
}
void CCyclicSystem_SetStateProc(This,BYTE byStateProc)
{
     //DECLARE_SINGLE_OPEN(CCyclicSystem)
	 DECLARE_SINGLE_OPEN(CCyclicSystem)
	 pT->m_byStateProc = byStateProc;
}
void CCyclicSystem_SetPeriod(This,BYTE byPeriod)
{
     //DECLARE_SINGLE_OPEN(CCyclicSystem)
	 DECLARE_SINGLE_OPEN(CCyclicSystem)
	 pT->m_byPeriod = byPeriod;
}
BYTE CCyclicSystem_GetStateProc(This)
{
     //DECLARE_SINGLE_OPEN(CCyclicSystem)
	 DECLARE_SINGLE_OPEN(CCyclicSystem)
	 return pT->m_byStateProc;
}
void CCyclicSystem_SetName(This,SINT* chProcName)
{
     //DECLARE_SINGLE_OPEN(CCyclicSystem)
	 DECLARE_SINGLE_OPEN(CCyclicSystem)
     strcpy(pT->m_chProcName,chProcName);
}
void CCyclicSystem_SetBoxID(This,BYTE byID)
{
     //DECLARE_SINGLE_OPEN(CCyclicSystem)
	 DECLARE_SINGLE_OPEN(CCyclicSystem)
	 pT->m_byBoxID = byID;
}
BOOL CCyclicSystem_GetMessage(This)
{
	BOOL res = TRUE;
	DECLARE_SINGLE_OPEN(CCyclicSystem)
	if( pT->m_byBoxID!=0xff)
	//if( pT->m_byBoxID==7)
	if(FGET(pT->m_byBoxID,(BYTE*)&pT->m_nsMessage)!=0)
	pT->EventHandler(pC,&pT->m_nsMessage);
	return res;
}
BOOL CCyclicSystem_EventHandler(This,SMESSAGE *pMsg)
{
    DECLARE_SINGLE_OPEN(CCyclicSystem)
	return TRUE;
}
void CCyclicSystem_CyclicProc(This)
{
	//DECLARE_SINGLE_OPEN(CCyclicSystem)
	DECLARE_SINGLE_OPEN(CCyclicSystem)
}
void CCyclicSystem_SendMessageData(This,BYTE byBox,BYTE byFor,BYTE byType,PVOID pData,WORD wLen)
{
    DECLARE_SINGLE_OPEN(CCyclicSystem)
	SMESSAGE m_sMsg;
	m_sMsg.m_swLen        = 9+wLen;
	m_sMsg.m_sbyFrom      = byFor;
	m_sMsg.m_sbyFor       = byFor;
	m_sMsg.m_sbyIntType   = 0;
	m_sMsg.m_sbyServerID  = 0;
	m_sMsg.m_sbyType      = byType;
	m_sMsg.m_sbyDirection = 0;
	m_sMsg.m_sbySensor    = 0;
	memcpy(&m_sMsg.m_sbyInfo[0],pData,wLen);
	FPUT(byBox,(BYTE*)&m_sMsg);
	return TRUE;
}
void CCyclicSystem_SendMessageData1(This,BYTE byBox,BYTE byFor,BYTE byType,SMESSAGE *pInMsg, PVOID pData,WORD wLen)
{
    DECLARE_SINGLE_OPEN(CCyclicSystem)
	pInMsg->m_swLen        = 9+wLen;
	pInMsg->m_sbyFrom      = byFor;
	pInMsg->m_sbyFor       = byFor;
	pInMsg->m_sbyIntType   = 0;
	pInMsg->m_sbyServerID  = 0;
	pInMsg->m_sbyType      = byType;
	pInMsg->m_sbyDirection = 0;
	pInMsg->m_sbySensor    = 0;
	memcpy(&pInMsg->m_sbyInfo[0],pData,wLen);
	FPUT(byBox,(BYTE*)pInMsg);
	return TRUE;
}
WORD CCyclicSystem_GetWordParam(This,BYTE *pbyParam,BYTE *pbyOut)
{
    DECLARE_SINGLE_OPEN(CCyclicSystem)
    #ifndef WIN32
	pbyOut[0] = pbyParam[1];
	pbyOut[1] = pbyParam[0];
    #else
	pbyOut[0] = pbyParam[0];
	pbyOut[1] = pbyParam[1];
    #endif
	return (WORD)*((WORD*)pbyOut);
}
void CCyclicSystem_CCyclicSystem(This)
{
	DECLARE_SINGLE_OPEN(CCyclicSystem)
	DECLARE_REGISTRATION(CCyclicSystem,SetBoxID)
	DECLARE_REGISTRATION(CCyclicSystem,CyclicProc)
	DECLARE_REGISTRATION(CCyclicSystem,Create)
	DECLARE_REGISTRATION(CCyclicSystem,CreateSuspend)
	DECLARE_REGISTRATION(CCyclicSystem,Start)
	DECLARE_REGISTRATION(CCyclicSystem,Stop)
	DECLARE_REGISTRATION(CCyclicSystem,SetStateProc)
	DECLARE_REGISTRATION(CCyclicSystem,SetPeriod)
	DECLARE_REGISTRATION(CCyclicSystem,GetStateProc)
	DECLARE_REGISTRATION(CCyclicSystem,SetName)
	DECLARE_REGISTRATION(CCyclicSystem,EventHandler)
	DECLARE_REGISTRATION(CCyclicSystem,GetMessage)

	DECLARE_REGISTRATION(CCyclicSystem,SetMsgAuto)
	DECLARE_REGISTRATION(CCyclicSystem,GetStateList)
	DECLARE_REGISTRATION(CCyclicSystem,HandleTask)
	DECLARE_REGISTRATION(CCyclicSystem,HandleEvent)
	DECLARE_REGISTRATION(CCyclicSystem,SetState)
	DECLARE_REGISTRATION(CCyclicSystem,GetStateCode)
	DECLARE_REGISTRATION(CCyclicSystem,GetState)
	DECLARE_REGISTRATION(CCyclicSystem,SendMessageData)
	DECLARE_REGISTRATION(CCyclicSystem,SendMessageData1)
	DECLARE_REGISTRATION(CCyclicSystem,GetWordParam)
	pT->m_byBoxID = 0xff;
    pT->m_pvState = BadStateCC;
    pT->m_vState  = S_BAD;
}
void CCyclicSystem_DCCyclicSystem(This)
{
	//DECLARE_SINGLE_OPEN(CCyclicSystem)
	DECLARE_SINGLE_OPEN(CCyclicSystem)
}
//DECLARE_SINGLE_CREATE(CCyclicSystem)
DECLARE_SINGLE_CREATE(CCyclicSystem)
```

#### bnrdebug.c
```c
#include "bnrdebug.h"
#include <stdarg.h>
#include <string.h>
#include <stdio.h>
#include "bnrmessage.h"
#define LenBuf  1500
#define LenBuf2 50
BYTE    HEX[] = "0123456789ABCDEF";
BYTE    st1[]={2,'^'};
BYTE    st2[]={3,'~','\n'};
BYTE    Str[]="\nInfo: Error:";
SLMESSAGE *m_pDebMsg;
BYTE  *DebugBufO;
void Info (char * Format,...)

{
  int     a,l,i,j,m;
  va_list arg;
  BYTE    c, *cp;
  va_start (arg,Format);
  DebugBufO = &m_pDebMsg->m_sbyInfo[0];
  for(j=1,i=0;(c=Format[i]) !=0 ; i++)
  {
   if (c!='%')
   {
    if(j==LenBuf){
     j=OutFrame(j,DebugBufO);
    }
    DebugBufO[j++]=c;
   }
   else
    switch(Format[++i])
    {
     case 'a':  if(j+9 > LenBuf){
                 j=OutFrame(j,DebugBufO);
                }
                cp=va_arg(arg, BYTE *);
                c=*(cp+3);
                DebugBufO[j++]=HEX[(c>>4) & 0x0f];
                DebugBufO[j++]=HEX[c & 0x0f];
                c=*(cp+2);
                DebugBufO[j++]=HEX[(c>>4) & 0x0f];
                DebugBufO[j++]=HEX[c & 0x0f];
                DebugBufO[j++]=':';
                c=*(cp+1);
                DebugBufO[j++]=HEX[(c>>4) & 0x0f];
                DebugBufO[j++]=HEX[c & 0x0f];
                c=*cp;
                DebugBufO[j++]=HEX[(c>>4) & 0x0f];
                DebugBufO[j++]=HEX[c & 0x0f];
                break;
     case 's':  cp=va_arg(arg, BYTE *);
                while((c=*(cp++))!=0)
                {
                 if(j == LenBuf){
                  j=OutFrame(j,DebugBufO);
                 }
                 DebugBufO[j++]=c;
                }
                break;
     case 'm':
                 cp=va_arg(arg, BYTE*);
                c=l=*(cp++);
                if(j+3 > LenBuf){
                 j=OutFrame(j,DebugBufO);
                 DebugBufO[j++]='\n';
                }
                DebugBufO[j++]=HEX[(c>>4) & 0x0f];
                DebugBufO[j++]=HEX[c & 0x0f];
                DebugBufO[j++]='_';
                for (a=1,m=0; a<l; a++,m++)
                {
                 if(j+5 > LenBuf){
                  j=OutFrame(j,DebugBufO);
                  DebugBufO[j++]='\n';
                 }
                 if (m==2){
                  DebugBufO[j++]='_';
                  m=0;
                 }
                 c=*(cp++);
                 DebugBufO[j++]=HEX[(c>>4) & 0x0f];
                 DebugBufO[j++]=HEX[c & 0x0f];
                }
                break;
	  case 'M':
		        cp=va_arg(arg, BYTE*);
		        c=*cp;
		        l=*(WORD*)(cp++);
		        if(j+3 > LenBuf){
			    j=OutFrame(j,DebugBufO);
			    DebugBufO[j++]='\n';
				}
				DebugBufO[j++]=HEX[(c>>4) & 0x0f];
				DebugBufO[j++]=HEX[c & 0x0f];
				DebugBufO[j++]='_';
				for (a=1,m=0; a<l; a++,m++)
				{
				if(j+5 > LenBuf){
				j=OutFrame(j,DebugBufO);
				DebugBufO[j++]='\n';
				}
				if (m==2){
				 DebugBufO[j++]='_';
				 m=0;
				}
				c=*(cp++);
				DebugBufO[j++]=HEX[(c>>4) & 0x0f];
				DebugBufO[j++]=HEX[c & 0x0f];
				}
                break;
     case 'w':  if(j+4 > LenBuf){
                 j=OutFrame(j,DebugBufO);
                }
                cp=va_arg(arg, BYTE*);
                c=*(cp+1);
                DebugBufO[j++]=HEX[(c>>4) & 0x0f];
                DebugBufO[j++]=HEX[c & 0x0f];
                c=*cp;
                DebugBufO[j++]=HEX[(c>>4) & 0x0f];
                DebugBufO[j++]=HEX[c & 0x0f];
                break;
     case 'b':  if(j+2 > LenBuf){
                 j=OutFrame(j,DebugBufO);
                }
                cp=va_arg(arg, BYTE *);
                c=*cp;
                DebugBufO[j++]=HEX[(c>>4) & 0x0f];
                DebugBufO[j++]=HEX[c & 0x0f];
                break;
     case 'd':  if(j+8 > LenBuf){
                 j=OutFrame(j,DebugBufO);
                }
                cp=va_arg(arg, BYTE *);
                c=*(cp+3);
                DebugBufO[j++]=HEX[(c>>4) & 0x0f];
                DebugBufO[j++]=HEX[c & 0x0f];
                c=*(cp+2);
                DebugBufO[j++]=HEX[(c>>4) & 0x0f];
                DebugBufO[j++]=HEX[c & 0x0f];
                c=*(cp+1);
                DebugBufO[j++]=HEX[(c>>4) & 0x0f];
                DebugBufO[j++]=HEX[c & 0x0f];
                c=*cp;
                DebugBufO[j++]=HEX[(c>>4) & 0x0f];
                DebugBufO[j++]=HEX[c & 0x0f];
                break;
     default :  j=1;
                for(i=0; Str[i]; i++)
                 DebugBufO[j++]=Str[i];
                DebugBufO[j++]='\"';
                for(i=0,a=1; Format[i]; i++){
                 if(Format[i]==0xa){
                  DebugBufO[j++]='\\';
                  DebugBufO[j++]='n';
                  a=0;
                 }
                 if(Format[i]==0xd){
                  DebugBufO[j++]='\\';
                  DebugBufO[j++]='r';
                  a=0;
                 }
                 if(a)
                  DebugBufO[j++]=Format[i];
                 else
                  a=1;
                }
                DebugBufO[j++]='\"';
                DebugBufO[0]=j;
                //FPUT(0x81,DebugBufO);
                return;
    }
  }
  OutFrame(j,DebugBufO);
  va_end(arg);
}
int OutFrame(int j, BYTE *DebugBufOf)
{
   m_pDebMsg->m_swLen        = j+9+1;
   m_pDebMsg->m_sbyFrom      = MDL_DEBMS;
   m_pDebMsg->m_sbyFor       = MDL_DEBMS;
   m_pDebMsg->m_sbyIntType   = 0;
   m_pDebMsg->m_sbyServerID  = 0;
   m_pDebMsg->m_sbyType      = EV_DEBMS_DEBOUT_IND;
   m_pDebMsg->m_sbyDirection = 0;
   m_pDebMsg->m_sbySensor    = 0;
   DebugBufO[0]   = 0x7e;
   DebugBufO[j]   = 0;
   #ifdef WIN32
   printf("%s",DebugBufO);
   #else
   DebugBufO[j] = 0x7e;
   FPUT(DEV_RSBUF_BOX_ID,(BYTE*)m_pDebMsg);
   #endif
   return 1;
}
```

#### bnrdigsensor.c
```c
/********************************************************************
 * COPYRIGHT -- Kontora
 ********************************************************************
 * Program: bnrmain
 * File: bnrlsens.c
 * Author: Abramenya
 * Created: January 19, 2009
 *******************************************************************/

#include "bnrdigsensor.h"
#ifdef _DEFAULT_INCLUDES
 #include <AsDefault.h>
#endif
#if MYSYSTEM_ID != 5
IMPORT_TASKCHAIN(Skip);
//пустое состояние
IMPORT_STATE(BadState);
//Обработчик событий дискретного датчика
//Digital Sensor Logic///////////////////////////////////////
DECLARE_TASKCHAIN(EvMcSetIn00){/*CMD_SETSTATE,SNS_STATE_FREE,*/EXIT_D,};
DECLARE_TASKCHAIN(EvMcRemIn00){/*CMD_SETSTATE,SNS_STATE_FREE,*/EXIT_D,};
DECLARE_TASKCHAIN(EvMcSetIn01){EXIT_D,};
DECLARE_TASKCHAIN(EvMcRemIn01){EXIT_D,};
DECLARE_TASKCHAIN(EvMcSetIn02){EXIT_D,};
DECLARE_TASKCHAIN(EvMcRemIn02){EXIT_D,};
DECLARE_TASKCHAIN(EvMcSetIn03){EXIT_D,};
DECLARE_TASKCHAIN(EvMcRemIn03){EXIT_D,};
DECLARE_TASKCHAIN(EvMcSetIn04){EXIT_D,};
DECLARE_TASKCHAIN(EvMcRemIn04){EXIT_D,};
DECLARE_TASKCHAIN(EvMcSetIn05){EXIT_D,};
DECLARE_TASKCHAIN(EvMcRemIn05){EXIT_D,};
DECLARE_TASKCHAIN(EvMcSetIn06){EXIT_D,};
DECLARE_TASKCHAIN(EvMcRemIn06){EXIT_D,};
DECLARE_TASKCHAIN(EvMcSetIn07){EXIT_D,};
DECLARE_TASKCHAIN(EvMcRemIn07){EXIT_D,};
DECLARE_TASKCHAIN(EvMcSetIn08){EXIT_D,};
DECLARE_TASKCHAIN(EvMcRemIn08){EXIT_D,};
DECLARE_TASKCHAIN(EvMcSetIn09){EXIT_D,};
DECLARE_TASKCHAIN(EvMcRemIn09){EXIT_D,};
/*DECLARE_TASKCHAIN(EvMcSetIn10){EXIT_D,};
DECLARE_TASKCHAIN(EvMcRemIn10){EXIT_D,};
DECLARE_TASKCHAIN(EvMcSetIn11){EXIT_D,};
DECLARE_TASKCHAIN(EvMcRemIn11){EXIT_D,};
DECLARE_TASKCHAIN(EvMcSetIn12){EXIT_D,};
DECLARE_TASKCHAIN(EvMcRemIn12){EXIT_D,};
DECLARE_TASKCHAIN(EvMcSetIn13){EXIT_D,};
DECLARE_TASKCHAIN(EvMcRemIn13){EXIT_D,};
DECLARE_TASKCHAIN(EvMcSetIn14){EXIT_D,};
DECLARE_TASKCHAIN(EvMcRemIn14){EXIT_D,};
DECLARE_TASKCHAIN(EvMcSetIn15){EXIT_D,};
DECLARE_TASKCHAIN(EvMcRemIn15){EXIT_D,};
DECLARE_TASKCHAIN(EvMcSetIn16){EXIT_D,};
DECLARE_TASKCHAIN(EvMcRemIn16){EXIT_D,};
DECLARE_TASKCHAIN(EvMcSetIn17){EXIT_D,};
DECLARE_TASKCHAIN(EvMcRemIn17){EXIT_D,};
DECLARE_TASKCHAIN(EvMcSetIn18){EXIT_D,};
DECLARE_TASKCHAIN(EvMcRemIn18){EXIT_D,};
DECLARE_TASKCHAIN(EvMcSetIn19){EXIT_D,};
DECLARE_TASKCHAIN(EvMcRemIn19){EXIT_D,};*/
DECLARE_STATE(Dig00StateFree)
{
    { EV_MCSET_IN00,          EvMcSetIn00},
	{ EV_MCREM_IN00,          EvMcRemIn00},
    { EV_MCSET_IN01,          EvMcSetIn01},
	{ EV_MCREM_IN01,          EvMcRemIn01},
    { EV_MCSET_IN02,          EvMcSetIn02},
	{ EV_MCREM_IN02,          EvMcRemIn02},
    { EV_MCSET_IN03,          EvMcSetIn03},
	{ EV_MCREM_IN03,          EvMcRemIn03},
    { EV_MCSET_IN04,          EvMcSetIn04},
	{ EV_MCREM_IN04,          EvMcRemIn04},
    { EV_MCSET_IN05,          EvMcSetIn05},
	{ EV_MCREM_IN05,          EvMcRemIn05},
    { EV_MCSET_IN06,          EvMcSetIn06},
	{ EV_MCREM_IN06,          EvMcRemIn06},
    { EV_MCSET_IN07,          EvMcSetIn07},
	{ EV_MCREM_IN07,          EvMcRemIn07},
    { EV_MCSET_IN08,          EvMcSetIn08},
	{ EV_MCREM_IN08,          EvMcRemIn08},
    { EV_MCSET_IN09,          EvMcSetIn09},
	{ EV_MCREM_IN09,          EvMcRemIn09},
    /*{ EV_MCSET_IN10,          EvMcSetIn10},
	{ EV_MCREM_IN10,          EvMcRemIn10},
    { EV_MCSET_IN11,          EvMcSetIn11},
	{ EV_MCREM_IN11,          EvMcRemIn11},
    { EV_MCSET_IN12,          EvMcSetIn12},
	{ EV_MCREM_IN12,          EvMcRemIn12},
    { EV_MCSET_IN13,          EvMcSetIn13},
	{ EV_MCREM_IN13,          EvMcRemIn13},
    { EV_MCSET_IN14,          EvMcSetIn14},
	{ EV_MCREM_IN14,          EvMcRemIn14},
    { EV_MCSET_IN15,          EvMcSetIn15},
	{ EV_MCREM_IN15,          EvMcRemIn15},
    { EV_MCSET_IN16,          EvMcSetIn16},
	{ EV_MCREM_IN16,          EvMcRemIn16},
    { EV_MCSET_IN17,          EvMcSetIn17},
	{ EV_MCREM_IN17,          EvMcRemIn17},
    { EV_MCSET_IN18,          EvMcSetIn18},
	{ EV_MCREM_IN18,          EvMcRemIn18},
    { EV_MCSET_IN19,          EvMcSetIn19},
	{ EV_MCREM_IN19,          EvMcRemIn19},*/
    { EV_UNKNOWN_REQ,         Skip       }
};
DECLARE_STATELIST(STL_DIGS00_SENS)
{
    { SNS_STATE_FREE,         Dig00StateFree     },
    { S_BAD,                  BadState           }
};
void CDigitalSensor_InitSensor(This,PVOID pParam)
{
     DECLARE_MULTI_OPEN(CDigitalSensor,CSensor)
	 BYTE i;
	 SSWITCHTABLE *pS = (SSWITCHTABLE*)pParam;
	 SDIGGATE *pDIN = pS->sSensorParamTable;
	 SDIGGATE *pDOT = pS->sOutGate[0];
	 pB->m_wAmInput  = pDIN->swAmpin;
	 pB->m_wAmOutput = pDOT->swAmpin;
	 New(sizeof(CPin*)*pB->m_wAmInput  ,pB->m_pINP);
	 New(sizeof(CPin*)*pB->m_wAmOutput ,pB->m_pOUT);
	 New(sizeof(BOOL*)*pB->m_wAmOutput ,pB->m_bINP);
	 New(sizeof(BOOL*)*pB->m_wAmOutput ,pB->m_bOUT);
	 New(sizeof(INT16*)*pB->m_wAmOutput,pB->m_nINP);
	 New(sizeof(INT16*)*pB->m_wAmOutput,pB->m_nOUT);
	 for (i=0;i<pB->m_wAmInput;i++)
	 {
	  pB->m_pINP[i]=0;
	  pB->m_bINP[i]=0;
	  pB->m_nINP[i]=0;
	 }
	 for (i=0;i<pB->m_wAmOutput;i++)
	 {
	  pT->m_nPulceTime[i] = 0;
	  pT->m_blPulceGo[i]  = FALSE;
	  pT->m_nCurrValue[i] = 0xffff;
	  pB->m_pOUT[i]=0;
	  pB->m_bOUT[i]=0;
	  pB->m_nOUT[i]=0;
	 }
	 pB->m_dwInState  = 0x00;
	 pB->m_dwOutState = 0;
     #ifdef DEB_CDigitalSensor
     Info("\n(%b)CDSNS::>Create Digital:In[%b]:Out[%b]",&pB->m_bySensorID,&pDIN->swAmpin,&pDOT->swAmpin);
     #endif
}
//INT _GLOBAL nOutDN,nOutUP,nNumber_D,nTime_D,nVal_D,nInC,nPS_GO,nPS_ST,nTM_STOP,nPL_OUT,n0_PL,n1_PL;
void CDigitalSensor_EventHandler(This,SMESSAGE *pMsg)
{
     DECLARE_MULTI_OPEN(CDigitalSensor,CSensor)
	 BYTE  byNumber;
	 UINT  wTime;
	 UINT  wValue;
	 switch (pMsg->m_sbyType)
	 {
	   case EV_SENSR_SET_DIGT_OUT_REQ:
		    byNumber = pMsg->m_sbyInfo[1];
			wValue   = pB->GetWordParam(pB,&pMsg->m_sbyInfo[2]);
			if(byNumber<pB->m_wAmOutput)
		    pT->SetRemOut(pT,byNumber,wValue);
	   break;
	   case EV_SENSR_SET_DIGT_PULCE_REQ:
		    byNumber = pMsg->m_sbyInfo[1];
			wTime    = pB->GetWordParam(pB,&pMsg->m_sbyInfo[2]);
			wValue   = pB->GetWordParam(pB,&pMsg->m_sbyInfo[4]);
			pT->SetPulce(pT,byNumber,wValue,wTime);
			//nNumber_D = byNumber;
			//nTime_D   = wTime;
			//nVal_D    = wValue;
			//nInC++;
	   break;
	   default:
	   break;
	 }
}
INT _GLOBAL nINrem;
void CDigitalSensor_SetPulce(This,BYTE byNumber,UINT wValue,UINT wTime)
{
     DECLARE_MULTI_OPEN(CDigitalSensor,CSensor)
	 pT->m_blPulceGo[byNumber]  = FALSE;
	 pT->m_nCurrValue[byNumber] = wValue;
	 if(wTime==0xffff)
	 {
 	  if(byNumber<pB->m_wAmOutput)
	  pT->SetRemOut(pT,byNumber,wValue);
	 }else
	 {
	  nINrem++;
 	  if(pT->m_nCurrValue[byNumber]==1)
	  {
	   #ifdef MY_MODEL
	   pB->m_dwInState  |= 1<<byNumber;
	   #endif
       pB->m_dwOutState |= 1<<byNumber;
	   *pB->m_bOUT[byNumber] = 1;

	  }
	  if(pT->m_nCurrValue[byNumber]==0)
	  {
	   #ifdef MY_MODEL
       pB->m_dwInState  &= ~(1<<byNumber);
	   #endif
	   pB->m_dwOutState &= ~(1<<byNumber);
	   *pB->m_bOUT[byNumber] = 0;
	  }
	  pT->m_blPulceGo[byNumber] = TRUE;
	  pT->m_nPulceTime[byNumber] = wTime/SYSTEM_QTIME;
	 }
}
void CDigitalSensor_SetRemOut(This,BYTE byNumber,UINT wValue)
{
     DECLARE_MULTI_OPEN(CDigitalSensor,CSensor)
	 CPin *pN;
	 pN = pB->m_pINP[byNumber];
     if (pN->m_byPinType==PIN_DG_INOT_BOL) *pB->m_bOUT[byNumber] = (BOOL)wValue;
     if (pN->m_byPinType==PIN_AN_INOT_INT) *pB->m_nOUT[byNumber] = wValue;
	 if (wValue)pB->m_dwOutState |= 1<<byNumber;else pB->m_dwOutState &= ~(1<<byNumber);
}
void CDigitalSensor_PreProc(This)
{
     DECLARE_MULTI_OPEN(CDigitalSensor,CSensor)
	 pT->EventGen(pT);
	 pT->PulceGen(pT);
}
void CDigitalSensor_PulceGen(This)
{
     DECLARE_MULTI_OPEN(CDigitalSensor,CSensor)
	 BYTE i;
	 for (i=0;i<pB->m_wAmOutput;i++)
	 if(pT->m_blPulceGo[i])
	 {
	  if(pT->m_nPulceTime[i]--==0)
	  {
	  if(pT->m_nCurrValue[i]==TRUE)
	  {
       pB->m_dwOutState &= ~(1<<i);
	   *pB->m_bOUT[i] = 0;
	  }
	  if(pT->m_nCurrValue[i]==FALSE)
	  {
	   pB->m_dwOutState |= 1<<i;
	   *pB->m_bOUT[i] = 1;
	  }
	  pT->m_blPulceGo[i] = FALSE;
	 }
	}
}
void CDigitalSensor_EventGen(This)
{
     DECLARE_MULTI_OPEN(CDigitalSensor,CSensor)
	 BYTE i,byState;
	 CPin *pN;
	 //nPL_GEN++;
     for (i=0;i<pB->m_wAmInput;i++)
	 {
	  pN = pB->m_pINP[i];
	  byState = pN->GetState(pN);
	  if(byState==PIN_STATE_ONN)
	  {
       #ifdef DEB_CDigitalSensor
	   //Info("\n(%b)CDSNS::>PIN[ON ] :L[%b]:S[%b]:P[%b]",&pB->m_bySensorID,&i,&pN->m_bySlotNumber,&pN->m_byPinNumber);
       #endif
	   pB->SetAutoEvent(pB,i+EV_MCSET_IN00);
	   pB->m_dwInState |= 1<<i;
	  }
	  if(byState==PIN_STATE_OFF)
	  {
       #ifdef DEB_CDigitalSensor
	   //Info("\n(%b)CDSNS::>PIN[OFF] :L[%b]:S[%b]:P[%b]",&pB->m_bySensorID,&i,&pN->m_bySlotNumber,&pN->m_byPinNumber);
       #endif
	   pB->SetAutoEvent(pB,i+EV_MCREM_IN00);
	   pB->m_dwInState &= ~(1<<i);
	  }
	  if(byState==PIN_STATE_TRI){}
	 }
}
void CDigitalSensor_Processing(This)
{
     DECLARE_MULTI_OPEN(CDigitalSensor,CSensor)
}
void CDigitalSensor_PostProc(This)
{
     DECLARE_MULTI_OPEN(CDigitalSensor,CSensor)
}
void CDigitalSensor_RunAutomat(This)
{
     DECLARE_MULTI_OPEN(CDigitalSensor,CSensor)
}
void CDigitalSensor_CDigitalSensor(This)
{
     DECLARE_MULTI_OPEN(CDigitalSensor,CSensor)
	 DECLARE_REGISTRATION(CDigitalSensor,EventGen)
	 DECLARE_REGISTRATION(CDigitalSensor,SetRemOut)
	 DECLARE_REGISTRATION(CDigitalSensor,SetPulce)
	 DECLARE_REGISTRATION(CDigitalSensor,PulceGen)
	 DECLARE_VIRTUAL_FUNC(CDigitalSensor,InitSensor)
	 DECLARE_VIRTUAL_FUNC(CDigitalSensor,EventHandler)
	 DECLARE_VIRTUAL_FUNC(CDigitalSensor,PreProc)
	 DECLARE_VIRTUAL_FUNC(CDigitalSensor,Processing)
	 DECLARE_VIRTUAL_FUNC(CDigitalSensor,PostProc)
	 DECLARE_VIRTUAL_FUNC(CDigitalSensor,RunAutomat)
}
void CDigitalSensor_DCDigitalSensor(This)
{
	 DECLARE_MULTI_OPEN(CDigitalSensor,CSensor)
	 Delete(sizeof(CPin*)*pB->m_wAmInput  ,pB->m_pINP);
	 Delete(sizeof(CPin*)*pB->m_wAmOutput ,pB->m_pOUT);
	 Delete(sizeof(BOOL*)*pB->m_wAmOutput ,pB->m_bINP);
	 Delete(sizeof(BOOL*)*pB->m_wAmOutput ,pB->m_bOUT);
	 Delete(sizeof(INT16*)*pB->m_wAmOutput,pB->m_nINP);
	 Delete(sizeof(INT16*)*pB->m_wAmOutput,pB->m_nOUT);
}
DECLARE_MULTI_CREATE(CDigitalSensor,CSensor)
#endif
```
